Yaskawa INFORM job: DPRINT3D7.JBI

/JOB
//NAME DPRINT3D7
//POS
///NPOS 985,0,0,0,0,0
///TOOL 9
///POSTYPE PULSE
///PULSE
C00000=38331,58153,-103296,76545,-120383,-87250,0
C00001=38829,58071,-103540,76008,-120603,-87388,0
C00002=39135,58069,-103553,75698,-120771,-87432,0
C00003=39547,58102,-103468,75295,-121021,-87464,0
C00004=40049,58223,-103131,74838,-121386,-87436,0
C00005=40275,59096,-100656,75000,-122141,-86754,0
C00006=47985,53725,-116873,64386,-120957,-92528,0
C00007=47675,53509,-117561,64622,-120583,-92677,0
C00008=47512,53337,-118114,64720,-120319,-92811,0
C00009=47414,53155,-118707,64742,-120065,-92966,0
C00010=47387,52969,-119318,64686,-119830,-93137,0
C00011=47431,52787,-119922,64554,-119625,-93316,0
C00012=47549,52614,-120504,64346,-119454,-93499,0
C00013=47574,52593,-120575,64308,-119436,-93523,0
C00014=47628,52527,-120798,64219,-119373,-93594,0
C00015=47840,52374,-121320,63916,-119254,-93772,0
C00016=48067,52268,-121685,63619,-119197,-93907,0
C00017=31263,52363,-120961,59625,-120633,-94164,0
C00018=30956,52566,-120274,60061,-120805,-93930,0
C00019=30684,52688,-119859,60420,-120875,-93775,0
C00020=30370,52784,-119536,60811,-120890,-93639,0
C00021=30027,52848,-119318,61220,-120850,-93528,0
C00022=29664,52879,-119210,61633,-120758,-93444,0
C00023=29293,52875,-119218,62038,-120617,-93392,0
C00024=29245,52869,-119235,62089,-120591,-93390,0
C00025=29099,52864,-119249,62246,-120531,-93372,0
C00026=28731,52813,-119411,62626,-120330,-93365,0
C00027=28447,52743,-119639,62904,-120137,-93388,0
C00028=23605,59262,-99913,71173,-124359,-87087,0
C00029=24011,59446,-99401,70849,-124736,-87010,0
C00030=24270,59629,-98895,70675,-125027,-86912,0
C00031=24478,59852,-98276,70574,-125325,-86774,0
C00032=24629,60106,-97571,70549,-125613,-86602,0
C00033=24674,60248,-97179,70575,-125751,-86501,0
C00034=24716,60482,-96534,70652,-125958,-86328,0
C00035=24702,60771,-95739,70814,-126174,-86103,0
C00036=24621,61063,-94936,71047,-126350,-85865,0
C00037=28498,55123,-112076,85369,-113238,-88875,0
C00038=37681,59282,-100081,77670,-120764,-86229,0
C00039=37996,59009,-100854,77242,-120771,-86495,0
C00040=38275,58852,-101304,76897,-120827,-86663,0
C00041=38591,58743,-101619,76535,-120935,-86797,0
C00042=38928,58687,-101786,76172,-121088,-86891,0
C00043=39106,58685,-101794,75993,-121188,-86918,0
C00044=39389,58708,-101735,75719,-121365,-86940,0
C00045=39717,58789,-101511,75424,-121607,-86921,0
C00046=40017,58920,-101147,75180,-121870,-86858,0
C00047=40209,59050,-100782,75046,-122072,-86781,0
C00048=48256,52888,-119608,63698,-120051,-93341,0
C00049=48323,52793,-119927,63580,-119956,-93441,0
C00050=48337,52781,-119967,63559,-119947,-93454,0
C00051=48383,52725,-120153,63482,-119894,-93514,0
C00052=48503,52640,-120443,63311,-119827,-93613,0
C00053=48657,52567,-120690,63107,-119789,-93704,0
C00054=48843,52511,-120885,62876,-119781,-93786,0
C00055=49053,52474,-121016,62628,-119806,-93852,0
C00056=49530,52439,-121146,62087,-119926,-93955,0
C00057=30578,51713,-123173,60079,-119485,-94678,0
C00058=30592,51957,-122328,60177,-119839,-94445,0
C00059=30557,52051,-122006,60259,-119958,-94350,0
C00060=30547,52064,-121961,60277,-119974,-94336,0
C00061=30518,52123,-121760,60336,-120045,-94277,0
C00062=30431,52212,-121454,60474,-120140,-94179,0
C00063=30313,52291,-121186,60642,-120207,-94088,0
C00064=30163,52358,-120957,60839,-120246,-94002,0
C00065=29988,52410,-120777,61056,-120257,-93927,0
C00066=29796,52445,-120656,61284,-120236,-93866,0
C00067=29593,52462,-120596,61515,-120187,-93820,0
C00068=29386,52460,-120600,61742,-120110,-93791,0
C00069=29358,52457,-120610,61771,-120096,-93790,0
C00070=29234,52452,-120622,61905,-120047,-93776,0
C00071=29027,52424,-120713,62120,-119936,-93772,0
C00072=28832,52377,-120868,62313,-119804,-93789,0
C00073=28655,52311,-121087,62476,-119656,-93826,0
C00074=28506,52230,-121360,62602,-119496,-93883,0
C00075=28262,52031,-122031,62779,-119148,-94040,0
C00076=22525,59894,-98134,72576,-124225,-86409,0
C00077=23013,59805,-98387,72040,-124442,-86560,0
C00078=23209,59804,-98394,71841,-124555,-86594,0
C00079=23405,59836,-98307,71658,-124693,-86602,0
C00080=23465,59857,-98249,71607,-124744,-86596,0
C00081=23613,59925,-98061,71491,-124883,-86567,0
C00082=23766,60034,-97760,71390,-125056,-86508,0
C00083=23890,60167,-97394,71331,-125230,-86427,0
C00084=23981,60318,-96976,71315,-125400,-86325,0
C00085=23998,60372,-96827,71324,-125452,-86286,0
C00086=24026,60515,-96435,71368,-125577,-86181,0
C00087=24020,60684,-95968,71460,-125703,-86049,0
C00088=23975,60851,-95509,71589,-125803,-85913,0
C00089=23899,60999,-95103,71741,-125867,-85785,0
C00090=23790,61133,-94734,71919,-125901,-85664,0
C00091=23657,61244,-94431,72108,-125903,-85556,0
C00092=23222,61486,-93767,72664,-125812,-85295,0
C00093=38158,60313,-97216,77640,-121705,-85464,0
C00094=38179,59892,-98385,77438,-121451,-85805,0
C00095=38226,59733,-98827,77323,-121377,-85939,0
C00096=38312,59585,-99244,77175,-121331,-86071,0
C00097=38351,59542,-99365,77117,-121327,-86112,0
C00098=38467,59441,-99648,76958,-121330,-86209,0
C00099=38632,59347,-99915,76754,-121365,-86309,0
C00100=38817,59282,-100102,76542,-121429,-86388,0
C00101=39014,59248,-100201,76330,-121521,-86444,0
C00102=39081,59248,-100204,76264,-121560,-86455,0
C00103=39251,59262,-100167,76100,-121668,-86468,0
C00104=39442,59310,-100036,75931,-121812,-86457,0
C00105=39615,59387,-99824,75792,-121964,-86420,0
C00106=39764,59489,-99539,75689,-122122,-86359,0
C00107=39882,59612,-99198,75626,-122275,-86278,0
C00108=39967,59750,-98814,75604,-122420,-86180,0
C00109=40106,60176,-97632,75659,-122792,-85861,0
C00110=49445,53618,-117255,62738,-121392,-92853,0
C00111=48956,53536,-117508,63236,-121106,-92850,0
C00112=48781,53486,-117664,63403,-120980,-92868,0
C00113=48758,53476,-117695,63424,-120959,-92873,0
C00114=48651,53442,-117803,63524,-120877,-92888,0
C00115=48502,53371,-118031,63654,-120735,-92930,0
C00116=48381,53287,-118302,63747,-120587,-92989,0
C00117=48292,53192,-118608,63800,-120438,-93063,0
C00118=48241,53092,-118936,63809,-120297,-93148,0
C00119=48228,52989,-119273,63775,-120166,-93242,0
C00120=48242,52939,-119441,63736,-120109,-93291,0
C00121=48106,52817,-119840,63829,-119909,-93386,0
C00122=49490,53423,-117887,62596,-121169,-93036,0
C00123=49557,53418,-117905,62520,-121189,-93050,0
C00124=49691,53409,-117940,62368,-121227,-93081,0
C00125=49826,53399,-117976,62215,-121265,-93111,0
C00126=49900,53394,-117995,62132,-121285,-93127,0
C00127=49913,53392,-117999,62117,-121289,-93130,0
C00128=49925,53391,-118003,62102,-121291,-93133,0
C00129=49938,53390,-118008,62087,-121295,-93137,0
C00130=49951,53389,-118013,62072,-121298,-93140,0
C00131=49964,53388,-118017,62057,-121301,-93143,0
C00132=49977,53386,-118022,62042,-121305,-93146,0
C00133=49990,53385,-118026,62028,-121307,-93150,0
C00134=50003,53384,-118030,62013,-121311,-93153,0
C00135=50016,53382,-118034,61998,-121314,-93156,0
C00136=50030,53381,-118039,61983,-121318,-93159,0
C00137=50043,53380,-118042,61967,-121321,-93162,0
C00138=50056,53379,-118047,61952,-121324,-93165,0
C00139=50068,53378,-118052,61938,-121328,-93169,0
C00140=50080,53376,-118056,61924,-121330,-93172,0
C00141=50093,53375,-118061,61910,-121332,-93175,0
C00142=50105,53374,-118067,61896,-121336,-93178,0
C00143=50111,53373,-118068,61889,-121337,-93179,0
C00144=50120,53368,-118085,61876,-121335,-93186,0
C00145=50164,53345,-118162,61817,-121321,-93213,0
C00146=50208,53322,-118238,61758,-121308,-93241,0
C00147=50243,53302,-118302,61710,-121297,-93265,0
C00148=50270,53287,-118355,61672,-121286,-93283,0
C00149=50290,53273,-118397,61644,-121277,-93298,0
C00150=50310,53260,-118441,61615,-121268,-93313,0
C00151=50331,53247,-118484,61587,-121259,-93328,0
C00152=50351,53234,-118527,61558,-121250,-93343,0
C00153=50371,53221,-118570,61529,-121241,-93358,0
C00154=50385,53212,-118602,61509,-121232,-93369,0
C00155=50399,53202,-118635,61489,-121226,-93380,0
C00156=50413,53192,-118668,61469,-121218,-93391,0
C00157=50425,53182,-118700,61451,-121209,-93402,0
C00158=50438,53173,-118732,61433,-121201,-93413,0
C00159=50450,53163,-118765,61414,-121193,-93424,0
C00160=50463,53153,-118797,61396,-121185,-93435,0
C00161=50475,53143,-118830,61377,-121177,-93446,0
C00162=50488,53134,-118862,61359,-121169,-93457,0
C00163=50499,53125,-118892,61342,-121162,-93466,0
C00164=50509,53116,-118919,61327,-121154,-93475,0
C00165=50519,53108,-118947,61312,-121147,-93484,0
C00166=50526,53101,-118969,61301,-121142,-93491,0
C00167=50535,53094,-118993,61288,-121135,-93500,0
C00168=50543,53086,-119020,61275,-121128,-93508,0
C00169=50552,53078,-119048,61261,-121120,-93518,0
C00170=50546,53069,-119075,61263,-121107,-93524,0
C00171=50540,53060,-119104,61266,-121093,-93531,0
C00172=50534,53051,-119133,61269,-121080,-93538,0
C00173=50527,53042,-119164,61272,-121065,-93546,0
C00174=50520,53033,-119194,61275,-121051,-93553,0
C00175=50513,53023,-119225,61279,-121036,-93560,0
C00176=50506,53014,-119255,61282,-121021,-93568,0
C00177=50499,53005,-119286,61285,-121007,-93575,0
C00178=50492,52996,-119316,61288,-120992,-93583,0
C00179=50485,52986,-119347,61292,-120977,-93590,0
C00180=50478,52977,-119377,61295,-120964,-93598,0
C00181=50470,52968,-119408,61299,-120947,-93605,0
C00182=50461,52958,-119440,61304,-120933,-93613,0
C00183=50453,52948,-119472,61309,-120916,-93620,0
C00184=50444,52938,-119504,61314,-120900,-93628,0
C00185=50432,52927,-119543,61321,-120881,-93636,0
C00186=50421,52915,-119582,61328,-120861,-93646,0
C00187=50409,52903,-119621,61336,-120842,-93655,0
C00188=50397,52891,-119660,61343,-120822,-93664,0
C00189=50385,52879,-119698,61351,-120803,-93673,0
C00190=50373,52867,-119737,61358,-120782,-93682,0
C00191=50359,52855,-119779,61367,-120761,-93692,0
C00192=50344,52841,-119822,61377,-120738,-93701,0
C00193=50326,52826,-119873,61391,-120712,-93713,0
C00194=50303,52808,-119932,61408,-120681,-93726,0
C00195=50280,52790,-119990,61424,-120649,-93739,0
C00196=50258,52773,-120049,61441,-120618,-93752,0
C00197=50231,52753,-120114,61461,-120582,-93766,0
C00198=50191,52726,-120201,61492,-120534,-93784,0
C00199=50166,52711,-120252,61512,-120505,-93795,0
C00200=50160,52710,-120257,61519,-120500,-93795,0
C00201=50148,52707,-120265,61531,-120494,-93796,0
C00202=50136,52704,-120273,61543,-120486,-93797,0
C00203=50124,52702,-120281,61555,-120477,-93797,0
C00204=50112,52699,-120290,61566,-120471,-93798,0
C00205=50100,52697,-120298,61579,-120463,-93798,0
C00206=50089,52694,-120305,61590,-120456,-93799,0
C00207=50079,52692,-120312,61600,-120450,-93799,0
C00208=50068,52690,-120319,61611,-120443,-93800,0
C00209=50057,52688,-120326,61622,-120436,-93800,0
C00210=50045,52686,-120332,61634,-120429,-93800,0
C00211=49900,52663,-120404,61783,-120350,-93799,0
C00212=49755,52641,-120475,61933,-120269,-93798,0
C00213=49610,52619,-120545,62083,-120189,-93797,0
C00214=30191,51747,-123046,60523,-119408,-94589,0
C00215=30111,51679,-123283,60580,-119283,-94644,0
C00216=30030,51611,-123519,60638,-119159,-94700,0
C00217=29986,51574,-123646,60670,-119093,-94730,0
C00218=29979,51568,-123665,60675,-119082,-94734,0
C00219=29971,51563,-123685,60681,-119072,-94738,0
C00220=29964,51558,-123703,60687,-119062,-94742,0
C00221=29957,51552,-123723,60692,-119051,-94747,0
C00222=29949,51547,-123741,60698,-119042,-94751,0
C00223=29942,51541,-123759,60703,-119032,-94756,0
C00224=29935,51536,-123779,60709,-119021,-94760,0
C00225=29927,51530,-123797,60715,-119011,-94765,0
C00226=29920,51525,-123817,60720,-119001,-94769,0
C00227=29913,51519,-123835,60726,-118990,-94773,0
C00228=29905,51514,-123855,60732,-118980,-94777,0
C00229=29898,51509,-123873,60737,-118971,-94781,0
C00230=29891,51504,-123892,60743,-118961,-94785,0
C00231=29884,51499,-123908,60748,-118951,-94789,0
C00232=29877,51494,-123925,60754,-118942,-94793,0
C00233=29869,51489,-123941,60760,-118933,-94797,0
C00234=29866,51487,-123949,60763,-118928,-94799,0
C00235=29852,51484,-123959,60776,-118920,-94800,0
C00236=29791,51472,-124001,60838,-118882,-94803,0
C00237=29730,51460,-124042,60900,-118846,-94807,0
C00238=29679,51450,-124075,60952,-118816,-94809,0
C00239=29638,51443,-124100,60994,-118792,-94811,0
C00240=29605,51438,-124116,61028,-118774,-94811,0
C00241=29572,51433,-124132,61063,-118757,-94812,0
C00242=29539,51429,-124149,61097,-118739,-94812,0
C00243=29506,51424,-124165,61131,-118722,-94812,0
C00244=29473,51419,-124182,61165,-118704,-94813,0
C00245=29449,51416,-124192,61191,-118692,-94812,0
C00246=29424,51413,-124202,61217,-118680,-94812,0
C00247=29400,51410,-124212,61242,-118668,-94812,0
C00248=29376,51407,-124220,61268,-118656,-94810,0
C00249=29352,51405,-124227,61293,-118646,-94810,0
C00250=29328,51403,-124235,61318,-118634,-94809,0
C00251=29305,51400,-124243,61344,-118623,-94808,0
C00252=29281,51398,-124251,61369,-118612,-94807,0
C00253=29257,51396,-124259,61394,-118601,-94806,0
C00254=29235,51394,-124266,61417,-118592,-94805,0
C00255=29215,51392,-124272,61439,-118583,-94804,0
C00256=29195,51390,-124278,61460,-118573,-94803,0
C00257=29179,51389,-124281,61477,-118566,-94802,0
C00258=29161,51388,-124285,61496,-118560,-94801,0
C00259=29142,51387,-124289,61517,-118551,-94799,0
C00260=29122,51385,-124293,61538,-118543,-94798,0
C00261=29101,51393,-124265,61565,-118548,-94787,0
C00262=29086,51399,-124246,61584,-118550,-94780,0
C00263=29071,51404,-124225,61603,-118554,-94772,0
C00264=29055,51410,-124204,61623,-118557,-94764,0
C00265=29040,51416,-124182,61643,-118561,-94756,0
C00266=29025,51422,-124162,61662,-118564,-94748,0
C00267=29009,51428,-124141,61682,-118568,-94740,0
C00268=28994,51434,-124119,61702,-118571,-94732,0
C00269=28979,51440,-124098,61721,-118574,-94724,0
C00270=28963,51446,-124078,61741,-118578,-94716,0
C00271=28948,51451,-124056,61760,-118581,-94708,0
C00272=28932,51458,-124033,61781,-118586,-94699,0
C00273=28917,51465,-124009,61801,-118589,-94690,0
C00274=28901,51472,-123985,61822,-118594,-94682,0
C00275=28884,51479,-123957,61844,-118600,-94671,0
C00276=28865,51488,-123926,61868,-118607,-94660,0
C00277=28846,51497,-123894,61893,-118612,-94648,0
C00278=28828,51506,-123863,61918,-118619,-94637,0
C00279=28809,51515,-123832,61942,-118625,-94626,0
C00280=28791,51524,-123800,61966,-118632,-94614,0
C00281=28772,51532,-123769,61991,-118638,-94603,0
C00282=28752,51543,-123731,62018,-118647,-94590,0
C00283=28732,51554,-123694,62045,-118655,-94577,0
C00284=28706,51569,-123639,62081,-118668,-94557,0
C00285=28680,51584,-123585,62116,-118680,-94538,0
C00286=28654,51600,-123530,62152,-118693,-94520,0
C00287=28628,51615,-123476,62188,-118707,-94500,0
C00288=28597,51635,-123406,62230,-118724,-94476,0
C00289=28555,51667,-123295,62291,-118754,-94440,0
C00290=28555,51673,-123275,62294,-118762,-94433,0
C00291=28554,51679,-123254,62298,-118770,-94427,0
C00292=28554,51685,-123232,62301,-118778,-94422,0
C00293=28553,51691,-123211,62304,-118786,-94415,0
C00294=28553,51697,-123191,62307,-118794,-94409,0
C00295=28553,51703,-123170,62310,-118802,-94404,0
C00296=28552,51708,-123153,62313,-118809,-94398,0
C00297=28552,51713,-123134,62315,-118816,-94393,0
C00298=28552,51718,-123116,62317,-118824,-94388,0
C00299=28553,51724,-123096,62320,-118831,-94383,0
C00300=28559,51761,-122965,62330,-118885,-94346,0
C00301=28570,51831,-122724,62350,-118985,-94278,0
C00302=28581,51902,-122480,62370,-119084,-94211,0
C00303=28587,51937,-122360,62380,-119133,-94177,0
C00304=26988,56207,-108778,66138,-123397,-90126,0
C00305=27559,55476,-110984,65169,-122914,-90833,0
C00306=34385,54484,-114157,79150,-115754,-90039,0
C00307=35133,53863,-116128,78153,-115638,-90720,0
C00308=28153,54774,-113144,64187,-122418,-91528,0
C00309=28772,54099,-115260,63191,-121909,-92212,0
C00310=35909,53269,-118056,77124,-115507,-91394,0
C00311=36715,52701,-119942,76063,-115359,-92059,0
C00312=29489,53589,-116898,62162,-121584,-92777,0
C00313=29679,53591,-116893,61956,-121660,-92805,0
C00314=30389,53528,-117109,61146,-121854,-92975,0
C00315=30449,53516,-117148,61075,-121862,-92995,0
C00316=37553,52159,-121785,74968,-115195,-92717,0
C00317=32557,56236,-108783,60130,-125967,-91111,0
C00318=31344,53310,-117832,59990,-121933,-93322,0
C00319=31411,53289,-117902,59905,-121930,-93352,0
C00320=32489,53643,-116779,58887,-122791,-93223,0
C00321=33235,55545,-110873,59024,-125452,-91789,0
C00322=33580,55212,-111891,58471,-125194,-92120,0
C00323=34127,55436,-111218,57982,-125691,-92047,0
C00324=33632,54047,-115515,57822,-123745,-93081,0
C00325=34746,54472,-114200,56798,-124719,-92936,0
C00326=41514,51531,-124061,70453,-116003,-93828,0
C00327=42611,51965,-122576,69442,-116893,-93495,0
C00328=35832,54919,-112836,55815,-125714,-92788,0
C00329=45678,52142,-122048,66179,-118202,-93704,0
C00330=45685,52643,-120356,66395,-118810,-93209,0
C00331=45693,53257,-118329,66662,-119525,-92621,0
C00332=45700,53794,-116593,66900,-120126,-92121,0
C00333=44762,54321,-114897,68151,-120297,-91501,0
C00334=44638,51679,-123626,67113,-117264,-94046,0
C00335=43562,51238,-125158,68100,-116350,-94385,0
C00336=43855,54873,-113154,69373,-120456,-90871,0
C00337=42976,55449,-111365,70566,-120600,-90230,0
C00338=42574,51681,-123560,69364,-116551,-93790,0
C00339=41623,52167,-121858,70596,-116757,-93166,0
C00340=42126,56052,-109528,71730,-120734,-89579,0
C00341=41304,56680,-107641,72868,-120856,-88917,0
C00342=40707,52678,-120113,71792,-116945,-92533,0
C00343=39824,53213,-118325,72955,-117117,-91892,0
C00344=40507,57334,-105705,73979,-120965,-88245,0
C00345=39896,57870,-104139,74839,-121043,-87706,0
C00346=39759,57838,-104230,74965,-120944,-87714,0
C00347=39709,57834,-104241,75013,-120914,-87710,0
C00348=38973,53774,-116493,74084,-117275,-91241,0
C00349=38152,54361,-114618,75181,-117415,-90581,0
C00350=38839,57797,-104329,75882,-120413,-87619,0
C00351=38784,57798,-104326,75937,-120383,-87610,0
C00352=38125,57905,-104004,76648,-120097,-87430,0
C00353=38000,57947,-103882,76792,-120057,-87378,0
C00354=37361,54974,-112698,76248,-117543,-89913,0
C00355=36597,55613,-110732,77286,-117655,-89235,0
C00356=37083,57698,-104582,77613,-119379,-87467,0
C00357=36088,57176,-106077,78410,-118484,-87789,0
C00358=35597,55333,-111561,78209,-116954,-89374,0
C00359=35382,55525,-110973,78501,-116984,-89174,0
C00360=34626,55201,-111945,79159,-116380,-89388,0
C00361=35067,56678,-107520,79250,-117606,-88101,0
C00362=34023,56202,-108911,80133,-116743,-88407,0
C00363=26988,56207,-108778,66138,-123397,-90126,0
C00364=26438,56968,-106524,67097,-123870,-89408,0
C00365=32953,55749,-110251,81058,-115896,-88704,0
C00366=31858,55317,-111539,82026,-115065,-88994,0
C00367=25909,57758,-104221,68046,-124333,-88678,0
C00368=25407,58565,-101904,68972,-124779,-87946,0
C00369=25677,58848,-101106,68834,-125167,-87771,0
C00370=25959,59324,-99770,68784,-125726,-87448,0
C00371=26059,59657,-98840,68852,-126061,-87208,0
C00372=30505,54262,-114777,83075,-113747,-89879,0
C00373=30483,54351,-114498,83125,-113791,-89790,0
C00374=30737,54907,-112777,83035,-114252,-89276,0
C00375=36475,52909,-119246,76394,-115443,-91819,0
C00376=39287,53519,-117321,73649,-117178,-91527,0
C00377=37677,52791,-119666,75075,-115836,-92070,0
C00378=33817,55911,-109778,58572,-126132,-91613,0
C00379=41548,52077,-122164,70640,-116630,-93251,0
C00380=38066,54265,-114919,75233,-117295,-90662,0
C00381=37534,52314,-121259,75046,-115335,-92550,0
C00382=37535,52252,-121281,75054,-115355,-92528,0
C00383=23394,59896,-98012,71737,-124791,-86493,0
C00384=23307,59866,-98096,71810,-124718,-86502,0
C00385=23275,59856,-98122,71837,-124691,-86504,0
C00386=23229,59845,-98154,71878,-124656,-86506,0
C00387=23180,59837,-98176,71923,-124621,-86504,0
C00388=23118,59828,-98200,71981,-124579,-86500,0
C00389=23054,59822,-98215,72044,-124537,-86494,0
C00390=22961,59823,-98212,72138,-124483,-86478,0
C00391=22921,59825,-98206,72180,-124462,-86470,0
C00392=22873,59829,-98192,72231,-124436,-86458,0
C00393=22786,59845,-98148,72326,-124398,-86431,0
C00394=22744,59854,-98121,72373,-124381,-86417,0
C00395=22700,59867,-98087,72423,-124364,-86401,0
C00396=22631,59892,-98014,72505,-124343,-86369,0
C00397=22541,59936,-97893,72617,-124323,-86320,0
C00398=22471,59982,-97763,72710,-124316,-86272,0
C00399=22404,60033,-97623,72802,-124313,-86221,0
C00400=22346,60090,-97463,72888,-124321,-86167,0
C00401=22292,60151,-97293,72971,-124335,-86110,0
C00402=22281,60166,-97251,72989,-124340,-86096,0
C00403=22248,60218,-97109,73047,-124357,-86051,0
C00404=22210,60287,-96917,73119,-124385,-85991,0
C00405=22180,60370,-96689,73188,-124427,-85921,0
C00406=22165,60435,-96507,73236,-124466,-85868,0
C00407=22160,60475,-96397,73260,-124491,-85836,0
C00408=22158,60512,-96296,73280,-124517,-85807,0
C00409=22158,60589,-96084,73317,-124572,-85747,0
C00410=22162,60631,-95969,73333,-124605,-85715,0
C00411=22168,60666,-95875,73344,-124633,-85689,0
C00412=22186,60745,-95657,73365,-124701,-85631,0
C00413=22205,60799,-95509,73372,-124751,-85592,0
C00414=22228,60849,-95372,73374,-124801,-85557,0
C00415=22247,60890,-95261,73375,-124841,-85529,0
C00416=22269,60927,-95159,73371,-124881,-85504,0
C00417=22309,60984,-95005,73359,-124945,-85467,0
C00418=22337,61021,-94903,73350,-124989,-85443,0
C00419=22368,61055,-94812,73336,-125033,-85422,0
C00420=22417,61101,-94686,73310,-125095,-85395,0
C00421=22453,61133,-94599,73290,-125140,-85376,0
C00422=22491,61162,-94520,73266,-125184,-85360,0
C00423=22546,61197,-94426,73229,-125243,-85343,0
C00424=22589,61223,-94356,73199,-125287,-85330,0
C00425=22634,61245,-94296,73165,-125332,-85321,0
C00426=22654,61253,-94273,73150,-125349,-85318,0
C00427=22740,61286,-94185,73081,-125426,-85307,0
C00428=22808,61305,-94135,73022,-125481,-85304,0
C00429=22900,61322,-94090,72940,-125549,-85307,0
C00430=22969,61328,-94075,72874,-125596,-85315,0
C00431=23064,61328,-94075,72780,-125654,-85331,0
C00432=23119,61323,-94088,72723,-125685,-85344,0
C00433=23209,61312,-94120,72628,-125733,-85368,0
C00434=23286,61294,-94170,72541,-125767,-85396,0
C00435=23362,61271,-94234,72454,-125797,-85426,0
C00436=23434,61239,-94320,72366,-125819,-85463,0
C00437=23504,61204,-94418,72278,-125835,-85502,0
C00438=23568,61160,-94538,72192,-125842,-85547,0
C00439=23629,61113,-94667,72107,-125844,-85593,0
C00440=23683,61059,-94815,72027,-125837,-85644,0
C00441=23733,61002,-94971,71948,-125826,-85696,0
C00442=23774,60940,-95141,71875,-125805,-85751,0
C00443=23810,60876,-95317,71806,-125779,-85807,0
C00444=23835,60815,-95486,71750,-125747,-85859,0
C00445=23860,60739,-95694,71687,-125705,-85921,0
C00446=23871,60669,-95887,71640,-125659,-85977,0
C00447=23876,60622,-96015,71612,-125627,-86014,0
C00448=23878,60597,-96082,71597,-125610,-86033,0
C00449=23876,60526,-96278,71563,-125554,-86087,0
C00450=23870,60468,-96439,71539,-125507,-86131,0
C00451=23853,60385,-96668,71515,-125434,-86193,0
C00452=23834,60325,-96830,71505,-125377,-86235,0
C00453=23799,60249,-97041,71502,-125298,-86288,0
C00454=23766,60193,-97195,71507,-125236,-86326,0
C00455=23714,60125,-97384,71526,-125153,-86370,0
C00456=23667,60074,-97523,71548,-125087,-86401,0
C00457=23601,60017,-97682,71587,-125004,-86435,0
C00458=23541,59974,-97800,71625,-124937,-86458,0
C00459=23468,59932,-97916,71679,-124861,-86478,0
C00460=23393,59890,-98030,71734,-124787,-86498,0
C00461=35331,54513,-113922,78210,-116284,-90036,0
C00462=36294,54920,-112685,77364,-117050,-89763,0
C00463=40946,51800,-122908,71212,-116196,-93384,0
C00464=33828,55886,-109704,58589,-126201,-91572,0
C00465=35386,54467,-114067,78137,-116276,-90086,0
C00466=35602,55200,-111812,78184,-116919,-89424,0
C00467=36475,55591,-110642,77434,-117637,-89168,0
C00468=42173,51768,-123052,69869,-116605,-93562,0
C00469=33599,55210,-111743,58490,-125297,-92062,0
C00470=34231,54631,-113535,79390,-115843,-89806,0
C00471=35132,54999,-112418,78593,-116543,-89557,0
C00472=34897,55209,-111772,78911,-116575,-89336,0
C00473=35366,55411,-111167,78505,-116951,-89203,0
C00474=35548,55248,-111666,78257,-116925,-89373,0
C00475=36108,54971,-112524,77576,-116998,-89694,0
C00476=34832,55467,-110986,57257,-126113,-92098,0
C00477=36977,53692,-116543,53945,-124582,-93918,0
C00478=39300,53750,-116408,73761,-117469,-91225,0
C00479=44308,56417,-108340,69642,-122190,-89529,0
C00480=34851,55449,-111041,79046,-116720,-89110,0
C00481=32913,57439,-105115,81710,-116938,-87125,0
C00482=36071,54502,-113971,77439,-116627,-90128,0
C00483=40136,51777,-122967,72078,-115873,-93316,0
C00484=48422,53258,-118219,63727,-120668,-92946,0
C00485=48439,53269,-118186,63714,-120687,-92938,0
C00486=48516,53313,-118044,63650,-120769,-92909,0
C00487=48581,53344,-117946,63594,-120831,-92892,0
C00488=48673,53380,-117832,63510,-120910,-92873,0
C00489=48745,53403,-117759,63442,-120965,-92863,0
C00490=48847,53429,-117677,63342,-121035,-92855,0
C00491=48909,53441,-117639,63281,-121073,-92854,0
C00492=49019,53461,-117580,63169,-121138,-92854,0
C00493=49115,53471,-117549,63069,-121186,-92859,0
C00494=49212,53478,-117530,62966,-121232,-92869,0
C00495=49309,53478,-117531,62859,-121269,-92883,0
C00496=49406,53475,-117544,62752,-121303,-92901,0
C00497=49502,53466,-117577,62642,-121327,-92925,0
C00498=49596,53453,-117621,62533,-121346,-92952,0
C00499=49685,53434,-117685,62425,-121357,-92983,0
C00500=49773,53412,-117759,62319,-121362,-93017,0
C00501=49854,53384,-117850,62216,-121359,-93054,0
C00502=49931,53354,-117952,62117,-121350,-93095,0
C00503=49995,53321,-118057,62032,-121332,-93133,0
C00504=50066,53280,-118194,61933,-121307,-93182,0
C00505=50120,53239,-118330,61854,-121275,-93228,0
C00506=50153,53211,-118423,61804,-121252,-93259,0
C00507=50170,53196,-118472,61779,-121238,-93275,0
C00508=50210,53150,-118623,61712,-121196,-93323,0
C00509=50239,53111,-118749,61661,-121157,-93363,0
C00510=50271,53054,-118939,61599,-121095,-93419,0
C00511=50286,53011,-119079,61562,-121046,-93461,0
C00512=50294,52953,-119271,61525,-120974,-93515,0
C00513=50293,52909,-119417,61506,-120915,-93555,0
C00514=50278,52851,-119606,61495,-120836,-93606,0
C00515=50259,52807,-119752,61495,-120772,-93643,0
C00516=50222,52753,-119932,61510,-120688,-93688,0
C00517=50184,52710,-120073,61532,-120618,-93722,0
C00518=50126,52661,-120235,61572,-120534,-93759,0
C00519=50071,52622,-120364,61615,-120463,-93787,0
C00520=49995,52579,-120504,61679,-120381,-93815,0
C00521=49966,52565,-120551,61703,-120352,-93824,0
C00522=49923,52545,-120615,61742,-120311,-93836,0
C00523=49874,52527,-120674,61787,-120271,-93845,0
C00524=49812,52505,-120746,61845,-120220,-93856,0
C00525=49745,52484,-120814,61909,-120169,-93866,0
C00526=49642,52460,-120892,62011,-120102,-93873,0
C00527=49597,52451,-120923,62057,-120073,-93876,0
C00528=49541,52441,-120954,62115,-120041,-93876,0
C00529=49435,52428,-120996,62225,-119987,-93873,0
C00530=49382,52422,-121012,62280,-119961,-93870,0
C00531=49326,52418,-121024,62340,-119937,-93866,0
C00532=49233,52416,-121029,62441,-119902,-93854,0
C00533=49107,52419,-121015,62582,-119862,-93833,0
C00534=48999,52429,-120979,62706,-119837,-93807,0
C00535=48893,52443,-120930,62828,-119818,-93779,0
C00536=48793,52463,-120859,62948,-119809,-93744,0
C00537=48695,52486,-120779,63067,-119805,-93708,0
C00538=48674,52493,-120756,63093,-119806,-93699,0
C00539=48605,52516,-120676,63179,-119811,-93667,0
C00540=48520,52548,-120566,63288,-119822,-93623,0
C00541=48436,52591,-120419,63400,-119848,-93570,0
C00542=48379,52628,-120295,63480,-119873,-93527,0
C00543=48349,52651,-120217,63523,-119893,-93501,0
C00544=48325,52674,-120142,63561,-119911,-93476,0
C00545=48278,52721,-119982,63634,-119953,-93424,0
C00546=48257,52748,-119891,63669,-119980,-93396,0
C00547=48243,52771,-119816,63695,-120004,-93372,0
C00548=48216,52825,-119636,63750,-120060,-93317,0
C00549=48205,52863,-119509,63780,-120104,-93279,0
C00550=48200,52901,-119386,63802,-120149,-93244,0
C00551=48198,52931,-119286,63819,-120184,-93215,0
C00552=48201,52960,-119189,63830,-120222,-93188,0
C00553=48212,53006,-119039,63839,-120282,-93147,0
C00554=48222,53037,-118938,63843,-120323,-93119,0
C00555=48236,53066,-118842,63841,-120365,-93095,0
C00556=48264,53108,-118704,63830,-120427,-93060,0
C00557=48285,53138,-118608,63821,-120471,-93035,0
C00558=48311,53167,-118515,63806,-120515,-93013,0
C00559=48352,53204,-118395,63778,-120575,-92985,0
C00560=48365,53215,-118360,63770,-120594,-92977,0
C00561=48397,53262,-118207,63756,-120662,-92938,0
C00562=30428,52147,-121485,60486,-120164,-94162,0
C00563=30434,52142,-121505,60477,-120158,-94167,0
C00564=30467,52107,-121623,60424,-120122,-94205,0
C00565=30508,52051,-121815,60353,-120058,-94264,0
C00566=30527,52011,-121952,60313,-120009,-94305,0
C00567=30542,51955,-122141,60270,-119936,-94359,0
C00568=30545,51923,-122253,60253,-119891,-94391,0
C00569=30543,51869,-122436,60229,-119816,-94442,0
C00570=30529,51823,-122595,60223,-119745,-94484,0
C00571=30509,51777,-122753,60224,-119674,-94525,0
C00572=30475,51733,-122906,60241,-119600,-94563,0
C00573=30436,51690,-123054,60265,-119526,-94599,0
C00574=30384,51649,-123192,60304,-119451,-94630,0
C00575=30326,51611,-123325,60350,-119377,-94659,0
C00576=30257,51576,-123445,60410,-119304,-94683,0
C00577=30183,51543,-123557,60477,-119233,-94705,0
C00578=30100,51515,-123654,60555,-119166,-94720,0
C00579=30013,51490,-123741,60640,-119102,-94733,0
C00580=29919,51470,-123810,60734,-119042,-94740,0
C00581=29823,51452,-123870,60833,-118986,-94744,0
C00582=29722,51441,-123909,60939,-118936,-94741,0
C00583=29654,51435,-123928,61011,-118907,-94738,0
C00584=29619,51432,-123938,61049,-118890,-94735,0
C00585=29515,51428,-123949,61162,-118851,-94725,0
C00586=29430,51427,-123951,61256,-118822,-94715,0
C00587=29306,51431,-123935,61394,-118787,-94694,0
C00588=29217,51437,-123911,61495,-118768,-94675,0
C00589=29101,51451,-123858,61630,-118750,-94645,0
C00590=29015,51466,-123805,61731,-118742,-94618,0
C00591=28909,51490,-123718,61860,-118742,-94579,0
C00592=28829,51513,-123638,61957,-118747,-94546,0
C00593=28737,51546,-123520,62074,-118763,-94501,0
C00594=28668,51576,-123415,62164,-118781,-94462,0
C00595=28594,51617,-123271,62264,-118813,-94411,0
C00596=28538,51653,-123144,62341,-118845,-94367,0
C00597=28484,51700,-122980,62422,-118890,-94314,0
C00598=28467,51717,-122922,62449,-118908,-94294,0
C00599=28445,51742,-122834,62485,-118934,-94267,0
C00600=28428,51769,-122741,62516,-118965,-94238,0
C00601=28408,51803,-122623,62553,-119004,-94202,0
C00602=28393,51839,-122499,62586,-119048,-94165,0
C00603=28384,51892,-122317,62620,-119116,-94112,0
C00604=28383,51915,-122239,62632,-119146,-94089,0
C00605=28385,51943,-122144,62643,-119184,-94062,0
C00606=28398,51994,-121970,62651,-119256,-94015,0
C00607=28407,52018,-121886,62652,-119292,-93992,0
C00608=28420,52044,-121798,62650,-119331,-93969,0
C00609=28440,52073,-121701,62641,-119375,-93944,0
C00610=28456,52094,-121631,62633,-119409,-93927,0
C00611=28502,52141,-121470,62604,-119487,-93887,0
C00612=28561,52186,-121321,62560,-119567,-93853,0
C00613=28626,52229,-121177,62509,-119645,-93821,0
C00614=28701,52267,-121049,62444,-119724,-93795,0
C00615=28781,52304,-120927,62373,-119799,-93772,0
C00616=28871,52335,-120823,62289,-119872,-93755,0
C00617=28964,52364,-120729,62200,-119943,-93742,0
C00618=28987,52369,-120711,62177,-119959,-93740,0
C00619=29076,52388,-120648,62088,-120016,-93735,0
C00620=29167,52403,-120599,61995,-120067,-93735,0
C00621=29223,52410,-120579,61937,-120096,-93736,0
C00622=29274,52415,-120564,61883,-120120,-93740,0
C00623=29386,52422,-120542,61763,-120169,-93749,0
C00624=29465,52423,-120540,61676,-120199,-93760,0
C00625=29543,52421,-120546,61590,-120225,-93773,0
C00626=29603,52419,-120553,61524,-120244,-93784,0
C00627=29659,52415,-120568,61460,-120258,-93796,0
C00628=29702,52411,-120584,61410,-120267,-93806,0
C00629=29812,52397,-120633,61283,-120288,-93836,0
C00630=29904,52380,-120692,61174,-120297,-93866,0
C00631=30007,52355,-120775,61049,-120300,-93903,0
C00632=30087,52331,-120860,60948,-120296,-93939,0
C00633=30179,52297,-120974,60832,-120283,-93983,0
C00634=30247,52267,-121080,60742,-120265,-94022,0
C00635=30322,52226,-121218,60641,-120235,-94072,0
C00636=30376,52190,-121342,60564,-120204,-94114,0
C00637=30442,52147,-121485,60471,-120168,-94163,0
C00638=25183,55522,-110657,67769,-121953,-90344,0
C00639=36362,52582,-120147,76424,-115182,-92059,0
C00640=39661,59488,-99412,75825,-122113,-86283,0
C00641=39593,59449,-99522,75876,-122046,-86305,0
C00642=39522,59413,-99620,75931,-121981,-86323,0
C00643=39445,59385,-99696,75995,-121916,-86334,0
C00644=39394,59369,-99740,76039,-121876,-86340,0
C00645=39366,59362,-99761,76062,-121855,-86342,0
C00646=39285,59345,-99806,76136,-121796,-86344,0
C00647=39218,59334,-99835,76199,-121750,-86343,0
C00648=39119,59326,-99854,76294,-121686,-86334,0
C00649=39046,59327,-99852,76366,-121644,-86323,0
C00650=38950,59335,-99826,76466,-121593,-86302,0
C00651=38877,59348,-99790,76544,-121559,-86282,0
C00652=38785,59372,-99721,76646,-121521,-86249,0
C00653=38715,59396,-99651,76726,-121497,-86220,0
C00654=38632,59435,-99542,76825,-121473,-86176,0
C00655=38568,59471,-99438,76905,-121459,-86138,0
C00656=38496,59522,-99294,76997,-121451,-86086,0
C00657=38441,59569,-99162,77072,-121449,-86040,0
C00658=38384,59631,-98987,77156,-121454,-85982,0
C00659=38365,59654,-98923,77184,-121459,-85961,0
C00660=38340,59689,-98827,77224,-121466,-85930,0
C00661=38319,59726,-98724,77261,-121476,-85897,0
C00662=38293,59773,-98591,77307,-121491,-85855,0
C00663=38270,59824,-98450,77351,-121511,-85811,0
C00664=38248,59899,-98240,77406,-121545,-85747,0
C00665=38240,59932,-98147,77428,-121561,-85719,0
C00666=38233,59973,-98035,77452,-121583,-85686,0
C00667=38229,60048,-97827,77488,-121628,-85626,0
C00668=38229,60084,-97725,77504,-121652,-85596,0
C00669=38232,60123,-97617,77518,-121678,-85566,0
C00670=38240,60167,-97496,77530,-121711,-85532,0
C00671=38247,60199,-97409,77537,-121735,-85508,0
C00672=38270,60273,-97205,77546,-121794,-85452,0
C00673=38304,60344,-97009,77543,-121861,-85400,0
C00674=38344,60413,-96818,77535,-121929,-85351,0
C00675=38393,60477,-96642,77514,-121999,-85307,0
C00676=38447,60539,-96472,77489,-122071,-85266,0
C00677=38510,60594,-96322,77451,-122145,-85231,0
C00678=38577,60647,-96180,77409,-122218,-85200,0
C00679=38594,60657,-96151,77397,-122236,-85194,0
C00680=38660,60695,-96048,77349,-122300,-85174,0
C00681=38728,60727,-95962,77296,-122362,-85159,0
C00682=38771,60743,-95919,77262,-122399,-85152,0
C00683=38811,60755,-95886,77229,-122431,-85148,0
C00684=38899,60778,-95823,77153,-122500,-85143,0
C00685=38961,60789,-95796,77097,-122545,-85144,0
C00686=39024,60795,-95780,77038,-122588,-85148,0
C00687=39072,60799,-95769,76993,-122621,-85152,0
C00688=39118,60799,-95770,76948,-122648,-85159,0
C00689=39154,60798,-95775,76913,-122670,-85166,0
C00690=39245,60790,-95798,76819,-122722,-85185,0
C00691=39323,60775,-95840,76736,-122760,-85209,0
C00692=39412,60752,-95907,76639,-122800,-85241,0
C00693=39483,60725,-95982,76557,-122825,-85273,0
C00694=39565,60686,-96090,76459,-122852,-85315,0
C00695=39627,60649,-96194,76381,-122865,-85355,0
C00696=39698,60598,-96335,76288,-122876,-85405,0
C00697=39751,60551,-96466,76215,-122877,-85451,0
C00698=39810,60487,-96642,76127,-122871,-85510,0
C00699=39846,60440,-96772,76071,-122862,-85552,0
C00700=39894,60362,-96988,75988,-122839,-85621,0
C00701=39920,60306,-97144,75937,-122818,-85669,0
C00702=39947,60227,-97364,75873,-122782,-85737,0
C00703=39958,60179,-97496,75841,-122756,-85776,0
C00704=39972,60101,-97713,75792,-122711,-85841,0
C00705=39974,60031,-97906,75758,-122667,-85896,0
C00706=39971,59962,-98099,75730,-122617,-85951,0
C00707=39957,59893,-98289,75713,-122563,-86003,0
C00708=39938,59826,-98475,75701,-122506,-86054,0
C00709=39908,59761,-98655,75702,-122445,-86101,0
C00710=39873,59699,-98829,75708,-122382,-86146,0
C00711=39858,59679,-98885,75714,-122359,-86160,0
C00712=39829,59640,-98990,75726,-122315,-86186,0
C00713=39780,59585,-99145,75750,-122248,-86224,0
C00714=39724,59536,-99280,75784,-122183,-86254,0
C00715=39665,59469,-99466,75813,-122102,-86299,0
C00716=39665,59415,-99488,75823,-122118,-86281,0
C00717=23831,60832,-95318,71801,-125814,-85787,0
C00718=23834,60823,-95341,71793,-125810,-85794,0
C00719=23856,60761,-95510,71740,-125776,-85845,0
C00720=23876,60680,-95734,71679,-125727,-85911,0
C00721=23883,60617,-95906,71640,-125684,-85960,0
C00722=23885,60533,-96137,71596,-125622,-86025,0
C00723=23878,60473,-96301,71572,-125573,-86070,0
C00724=23858,60379,-96560,71546,-125489,-86139,0
C00725=23844,60334,-96683,71537,-125448,-86172,0
C00726=23819,60267,-96869,71528,-125381,-86220,0
C00727=23784,60203,-97045,71532,-125312,-86263,0
C00728=23744,60141,-97214,71541,-125242,-86304,0
C00729=23695,60085,-97369,71563,-125169,-86339,0
C00730=23641,60031,-97517,71591,-125097,-86371,0
C00731=23580,59984,-97646,71629,-125026,-86397,0
C00732=23515,59941,-97765,71673,-124955,-86420,0
C00733=23444,59905,-97863,71727,-124886,-86435,0
C00734=23371,59874,-97950,71786,-124819,-86448,0
C00735=23293,59850,-98013,71853,-124756,-86453,0
C00736=23214,59832,-98064,71925,-124695,-86454,0
C00737=23132,59822,-98089,72003,-124641,-86448,0
C00738=23050,59817,-98102,72083,-124588,-86438,0
C00739=22967,59821,-98090,72168,-124543,-86421,0
C00740=22886,59830,-98066,72255,-124502,-86401,0
C00741=22845,59836,-98046,72299,-124483,-86388,0
C00742=22792,59846,-98020,72357,-124459,-86372,0
C00743=22738,59860,-97979,72419,-124439,-86352,0
C00744=22687,59877,-97931,72479,-124421,-86330,0
C00745=22633,59898,-97874,72543,-124405,-86305,0
C00746=22586,59919,-97813,72601,-124394,-86280,0
C00747=22541,59945,-97742,72658,-124386,-86253,0
C00748=22490,59976,-97657,72724,-124379,-86221,0
C00749=22449,60005,-97574,72780,-124375,-86191,0
C00750=22412,60037,-97486,72832,-124378,-86160,0
C00751=22366,60079,-97370,72898,-124381,-86120,0
C00752=22335,60113,-97275,72946,-124388,-86088,0
C00753=22307,60150,-97172,72992,-124398,-86055,0
C00754=22270,60202,-97029,73054,-124414,-86008,0
C00755=22248,60240,-96923,73095,-124428,-85975,0
C00756=22229,60281,-96811,73133,-124447,-85940,0
C00757=22204,60341,-96644,73188,-124475,-85889,0
C00758=22191,60381,-96533,73220,-124497,-85855,0
C00759=22183,60424,-96416,73249,-124522,-85821,0
C00760=22173,60476,-96272,73283,-124555,-85779,0
C00761=22168,60532,-96119,73316,-124591,-85734,0
C00762=22171,60613,-95897,73352,-124651,-85672,0
C00763=22174,60647,-95805,73366,-124676,-85647,0
C00764=22180,60686,-95698,73379,-124709,-85618,0
C00765=22190,60727,-95584,73389,-124744,-85587,0
C00766=22206,60782,-95433,73401,-124793,-85547,0
C00767=22225,60837,-95282,73408,-124844,-85508,0
C00768=22273,60929,-95033,73405,-124938,-85445,0
C00769=22305,60980,-94893,73399,-124994,-85411,0
C00770=22317,60995,-94854,73394,-125012,-85402,0
C00771=22359,61043,-94723,73376,-125072,-85372,0
C00772=22418,61102,-94561,73347,-125150,-85336,0
C00773=22433,61115,-94528,73338,-125168,-85329,0
C00774=22484,61155,-94420,73307,-125228,-85307,0
C00775=22554,61203,-94289,73261,-125305,-85282,0
C00776=22630,61243,-94182,73206,-125380,-85264,0
C00777=22709,61278,-94087,73145,-125453,-85250,0
C00778=22729,61285,-94068,73128,-125472,-85249,0
C00779=22791,61304,-94019,73076,-125523,-85245,0
C00780=22858,61320,-93974,73018,-125576,-85244,0
C00781=22876,61324,-93963,73002,-125590,-85244,0
C00782=22920,61329,-93950,72961,-125620,-85248,0
C00783=22963,61332,-93942,72920,-125649,-85253,0
C00784=23049,61334,-93939,72835,-125704,-85266,0
C00785=23096,61331,-93947,72788,-125730,-85277,0
C00786=23136,61326,-93960,72745,-125752,-85287,0
C00787=23224,61312,-94000,72650,-125796,-85314,0
C00788=23285,61296,-94045,72582,-125821,-85336,0
C00789=23342,61276,-94098,72515,-125843,-85361,0
C00790=23387,61260,-94143,72462,-125859,-85381,0
C00791=23428,61241,-94195,72412,-125870,-85402,0
C00792=23457,61226,-94236,72375,-125877,-85419,0
C00793=23534,61181,-94359,72275,-125891,-85467,0
C00794=23594,61137,-94481,72193,-125896,-85512,0
C00795=23660,61079,-94639,72097,-125893,-85567,0
C00796=23709,61027,-94783,72022,-125884,-85616,0
C00797=23761,60960,-94967,71936,-125867,-85676,0
C00798=23797,60900,-95132,71869,-125844,-85729,0
C00799=23838,60825,-95335,71791,-125813,-85793,0
C00800=35332,54454,-113945,78218,-116301,-90015,0
C00801=36294,54861,-112707,77372,-117067,-89742,0
C00802=40946,51737,-122931,71220,-116218,-93362,0
C00803=33828,55829,-109726,58601,-126228,-91554,0
C00804=35386,54408,-114089,78145,-116292,-90065,0
C00805=35602,55142,-111834,78192,-116935,-89403,0
C00806=36475,55534,-110664,77442,-117653,-89148,0
C00807=42174,51704,-123075,69877,-116629,-93541,0
C00808=33600,55152,-111765,58501,-125325,-92044,0
C00809=34231,54572,-113557,79398,-115858,-89785,0
C00810=35133,54941,-112440,78601,-116559,-89536,0
C00811=34898,55151,-111794,78919,-116591,-89316,0
C00812=35366,55353,-111189,78513,-116967,-89183,0
C00813=35548,55190,-111688,78265,-116942,-89353,0
C00814=36108,54913,-112546,77584,-117015,-89673,0
C00815=34832,55409,-111009,57268,-126141,-92080,0
C00816=36963,53643,-116530,53978,-124624,-93889,0
C00817=39300,53691,-116430,73769,-117489,-91204,0
C00818=44279,56342,-108418,69675,-122178,-89522,0
C00819=34851,55391,-111063,79054,-116735,-89090,0
C00820=32925,57370,-105176,81701,-116951,-87118,0
C00821=36071,54444,-113993,77447,-116644,-90107,0
C00822=40136,51714,-122990,72085,-115895,-93295,0
C00823=48476,53281,-117971,63718,-120815,-92857,0
C00824=48534,53311,-117879,63668,-120872,-92840,0
C00825=48598,53340,-117786,63612,-120931,-92824,0
C00826=48615,53347,-117762,63596,-120946,-92819,0
C00827=48661,53363,-117714,63553,-120983,-92812,0
C00828=48707,53377,-117670,63510,-121018,-92807,0
C00829=48802,53402,-117591,63418,-121084,-92799,0
C00830=48855,53413,-117556,63366,-121118,-92797,0
C00831=48901,53421,-117531,63318,-121145,-92797,0
C00832=49007,53437,-117483,63210,-121205,-92799,0
C00833=49083,53444,-117462,63130,-121242,-92804,0
C00834=49157,53448,-117452,63051,-121275,-92813,0
C00835=49216,53451,-117445,62988,-121300,-92820,0
C00836=49272,53450,-117448,62927,-121321,-92829,0
C00837=49312,53449,-117453,62881,-121335,-92837,0
C00838=49422,53442,-117478,62757,-121368,-92860,0
C00839=49514,53431,-117516,62652,-121389,-92884,0
C00840=49619,53413,-117577,62527,-121407,-92918,0
C00841=49703,53393,-117644,62426,-121414,-92949,0
C00842=49798,53365,-117736,62308,-121416,-92989,0
C00843=49873,53337,-117829,62212,-121409,-93026,0
C00844=49958,53299,-117954,62100,-121393,-93074,0
C00845=50018,53266,-118063,62019,-121375,-93113,0
C00846=50088,53220,-118216,61920,-121343,-93166,0
C00847=50133,53182,-118339,61852,-121312,-93207,0
C00848=50184,53129,-118514,61770,-121263,-93263,0
C00849=50213,53089,-118643,61719,-121224,-93303,0
C00850=50248,53024,-118859,61650,-121153,-93368,0
C00851=50260,52992,-118964,61621,-121118,-93399,0
C00852=50273,52942,-119128,61583,-121058,-93447,0
C00853=50274,52892,-119293,61558,-120995,-93493,0
C00854=50268,52842,-119457,61540,-120928,-93537,0
C00855=50249,52793,-119618,61538,-120858,-93579,0
C00856=50224,52745,-119776,61543,-120787,-93620,0
C00857=50186,52699,-119928,61563,-120713,-93656,0
C00858=50143,52654,-120076,61590,-120638,-93691,0
C00859=50088,52612,-120212,61631,-120565,-93721,0
C00860=50027,52573,-120343,61679,-120492,-93748,0
C00861=49956,52537,-120458,61741,-120421,-93771,0
C00862=49880,52504,-120566,61808,-120351,-93790,0
C00863=49797,52476,-120657,61888,-120286,-93803,0
C00864=49709,52451,-120738,61972,-120222,-93813,0
C00865=49616,52432,-120800,62066,-120165,-93818,0
C00866=49521,52415,-120853,62163,-120110,-93819,0
C00867=49472,52409,-120874,62214,-120084,-93818,0
C00868=49408,52401,-120899,62281,-120051,-93816,0
C00869=49338,52395,-120916,62355,-120020,-93811,0
C00870=49271,52392,-120923,62427,-119993,-93804,0
C00871=49199,52391,-120928,62506,-119965,-93794,0
C00872=49133,52392,-120922,62580,-119943,-93784,0
C00873=49067,52395,-120907,62654,-119926,-93770,0
C00874=48991,52401,-120888,62740,-119906,-93754,0
C00875=48927,52408,-120861,62814,-119894,-93737,0
C00876=48867,52418,-120826,62885,-119885,-93719,0
C00877=48790,52432,-120777,62976,-119875,-93694,0
C00878=48734,52445,-120733,63043,-119872,-93674,0
C00879=48680,52460,-120680,63110,-119873,-93652,0
C00880=48607,52482,-120604,63200,-119875,-93620,0
C00881=48558,52500,-120543,63262,-119880,-93596,0
C00882=48513,52520,-120475,63321,-119890,-93570,0
C00883=48448,52551,-120371,63407,-119905,-93531,0
C00884=48409,52572,-120298,63459,-119919,-93505,0
C00885=48374,52596,-120218,63509,-119936,-93477,0
C00886=48332,52626,-120117,63569,-119958,-93443,0
C00887=48292,52659,-120006,63628,-119986,-93406,0
C00888=48247,52710,-119837,63701,-120032,-93352,0
C00889=48230,52731,-119765,63730,-120052,-93329,0
C00890=48213,52757,-119679,63760,-120079,-93302,0
C00891=48200,52786,-119585,63788,-120109,-93274,0
C00892=48184,52824,-119457,63823,-120150,-93236,0
C00893=48174,52864,-119327,63853,-120195,-93197,0
C00894=48173,52933,-119097,63886,-120280,-93132,0
C00895=48179,52974,-118964,63899,-120332,-93095,0
C00896=48203,53028,-118789,63897,-120406,-93049,0
C00897=48234,53081,-118617,63889,-120482,-93005,0
C00898=48278,53132,-118452,63864,-120560,-92964,0
C00899=48328,53182,-118292,63833,-120638,-92926,0
C00900=48410,53241,-118101,63771,-120742,-92884,0
C00901=48454,53322,-117841,63760,-120854,-92818,0
C00902=39622,59390,-99557,75854,-122076,-86295,0
C00903=39566,59365,-99627,75899,-122025,-86307,0
C00904=39518,59344,-99684,75938,-121984,-86316,0
C00905=39466,59327,-99732,75982,-121941,-86323,0
C00906=39409,59312,-99772,76032,-121898,-86326,0
C00907=39355,59300,-99806,76080,-121858,-86329,0
C00908=39302,59291,-99829,76130,-121821,-86327,0
C00909=39244,59286,-99843,76185,-121784,-86323,0
C00910=39203,59282,-99851,76225,-121758,-86320,0
C00911=39119,59281,-99854,76307,-121707,-86309,0
C00912=39036,59284,-99843,76391,-121661,-86294,0
C00913=38954,59296,-99809,76478,-121621,-86273,0
C00914=38873,59312,-99762,76566,-121584,-86249,0
C00915=38796,59337,-99690,76653,-121555,-86217,0
C00916=38721,59366,-99608,76740,-121530,-86183,0
C00917=38651,59403,-99503,76826,-121514,-86143,0
C00918=38585,59444,-99388,76909,-121501,-86101,0
C00919=38526,59491,-99253,76988,-121498,-86054,0
C00920=38471,59542,-99110,77064,-121498,-86005,0
C00921=38425,59599,-98951,77134,-121507,-85953,0
C00922=38383,59658,-98786,77201,-121521,-85899,0
C00923=38352,59722,-98608,77260,-121543,-85843,0
C00924=38325,59787,-98427,77314,-121569,-85787,0
C00925=38309,59855,-98238,77359,-121602,-85731,0
C00926=38302,59897,-98119,77385,-121625,-85696,0
C00927=38293,59993,-97854,77435,-121681,-85618,0
C00928=38295,60052,-97689,77459,-121720,-85571,0
C00929=38308,60134,-97464,77482,-121778,-85508,0
C00930=38324,60193,-97300,77492,-121825,-85462,0
C00931=38354,60272,-97085,77496,-121893,-85404,0
C00932=38385,60330,-96923,77492,-121950,-85362,0
C00933=38432,60401,-96729,77476,-122022,-85313,0
C00934=38476,60455,-96581,77457,-122083,-85277,0
C00935=38538,60517,-96413,77424,-122160,-85237,0
C00936=38594,60564,-96284,77390,-122224,-85208,0
C00937=38668,60614,-96148,77339,-122301,-85179,0
C00938=38735,60652,-96045,77291,-122367,-85159,0
C00939=38779,60671,-95992,77256,-122406,-85150,0
C00940=38834,60695,-95930,77213,-122454,-85140,0
C00941=38893,60715,-95875,77164,-122503,-85133,0
C00942=38982,60737,-95818,77087,-122572,-85129,0
C00943=39019,60744,-95799,77054,-122600,-85129,0
C00944=39063,60750,-95781,77014,-122631,-85130,0
C00945=39111,60754,-95774,76968,-122663,-85135,0
C00946=39175,60757,-95766,76907,-122705,-85142,0
C00947=39240,60756,-95770,76843,-122745,-85152,0
C00948=39351,60742,-95809,76728,-122805,-85180,0
C00949=39416,60730,-95843,76660,-122837,-85199,0
C00950=39498,60702,-95922,76566,-122869,-85234,0
C00951=39578,60670,-96012,76473,-122898,-85271,0
C00952=39653,60629,-96127,76381,-122917,-85315,0
C00953=39724,60583,-96253,76290,-122931,-85361,0
C00954=39788,60530,-96400,76203,-122936,-85413,0
C00955=39849,60474,-96557,76118,-122936,-85467,0
C00956=39899,60411,-96731,76039,-122925,-85524,0
C00957=39937,60359,-96874,75979,-122914,-85571,0
C00958=39946,60346,-96912,75963,-122910,-85583,0
C00959=39964,60310,-97010,75929,-122898,-85614,0
C00960=39979,60274,-97109,75898,-122883,-85644,0
C00961=40007,60199,-97318,75836,-122849,-85708,0
C00962=40019,60145,-97467,75799,-122821,-85752,0
C00963=40027,60090,-97618,75766,-122788,-85797,0
C00964=40032,60049,-97732,75743,-122764,-85830,0
C00965=40033,60011,-97839,75725,-122739,-85861,0
C00966=40031,59978,-97928,75712,-122716,-85886,0
C00967=40023,59900,-98146,75684,-122657,-85947,0
C00968=40010,59846,-98295,75673,-122614,-85988,0
C00969=39994,59797,-98431,75667,-122571,-86025,0
C00970=39979,59756,-98544,75663,-122534,-86055,0
C00971=39960,59718,-98649,75664,-122498,-86083,0
C00972=39927,59663,-98803,75673,-122440,-86122,0
C00973=39902,59625,-98908,75680,-122400,-86149,0
C00974=39875,59590,-99005,75692,-122360,-86173,0
C00975=39831,59543,-99135,75715,-122302,-86203,0
C00976=39798,59511,-99224,75732,-122261,-86224,0
C00977=39761,59480,-99309,75755,-122218,-86243,0
C00978=39709,59443,-99412,75791,-122162,-86265,0
C00979=39692,59432,-99444,75803,-122145,-86272,0
C00980=39621,59373,-99605,75848,-122063,-86308,0
C00981=29169,52326,-120674,61995,-120075,-93729,0
C00982=29228,52335,-120645,61935,-120109,-93730,0
C00983=29300,52345,-120612,61861,-120148,-93730,0
C00984=29377,52353,-120587,61780,-120186,-93735,0
//INST
///DATE 2025/02/20 16:20
///COMM Generated using RoboDK
///ATTR SC,RW
///GROUP1 RB1
NOP
MOVL C00000 V=60.0 PL=1
MOVL C00001 V=60.0 PL=1
MOVL C00002 V=60.0 PL=1
MOVL C00003 V=60.0 PL=1
MOVL C00004 V=60.0 PL=1
MOVL C00005 V=130.0 PL=1
MOVL C00006 V=60.0 PL=1
MOVL C00007 V=60.0 PL=1
MOVL C00008 V=60.0 PL=1
MOVL C00009 V=60.0 PL=1
MOVL C00010 V=60.0 PL=1
MOVL C00011 V=60.0 PL=1
MOVL C00012 V=60.0 PL=1
MOVL C00013 V=60.0 PL=1
MOVL C00014 V=60.0 PL=1
MOVL C00015 V=60.0 PL=1
MOVL C00016 V=60.0 PL=1
MOVL C00017 V=60.0 PL=1
MOVL C00018 V=60.0 PL=1
MOVL C00019 V=60.0 PL=1
MOVL C00020 V=60.0 PL=1
MOVL C00021 V=60.0 PL=1
MOVL C00022 V=60.0 PL=1
MOVL C00023 V=60.0 PL=1
MOVL C00024 V=60.0 PL=1
MOVL C00025 V=60.0 PL=1
MOVL C00026 V=60.0 PL=1
MOVL C00027 V=60.0 PL=1
MOVL C00028 V=60.0 PL=1
MOVL C00029 V=60.0 PL=1
MOVL C00030 V=60.0 PL=1
MOVL C00031 V=60.0 PL=1
MOVL C00032 V=60.0 PL=1
MOVL C00033 V=60.0 PL=1
MOVL C00034 V=60.0 PL=1
MOVL C00035 V=60.0 PL=1
MOVL C00036 V=60.0 PL=1
MOVL C00037 V=60.0 PL=1
MOVL C00038 V=60.0 PL=1
MOVL C00039 V=60.0 PL=1
MOVL C00040 V=60.0 PL=1
MOVL C00041 V=60.0 PL=1
MOVL C00042 V=60.0 PL=1
MOVL C00043 V=60.0 PL=1
MOVL C00044 V=60.0 PL=1
MOVL C00045 V=60.0 PL=1
MOVL C00046 V=60.0 PL=1
MOVL C00047 V=60.0 PL=1
MOVL C00048 V=130.0 PL=1
MOVL C00049 V=30.0 PL=1
MOVL C00050 V=30.0 PL=1
MOVL C00051 V=30.0 PL=1
MOVL C00052 V=30.0 PL=1
MOVL C00053 V=30.0 PL=1
MOVL C00054 V=30.0 PL=1
MOVL C00055 V=30.0 PL=1
MOVL C00056 V=30.0 PL=1
MOVL C00057 V=30.0 PL=1
MOVL C00058 V=30.0 PL=1
MOVL C00059 V=30.0 PL=1
MOVL C00060 V=30.0 PL=1
MOVL C00061 V=30.0 PL=1
MOVL C00062 V=30.0 PL=1
MOVL C00063 V=30.0 PL=1
MOVL C00064 V=30.0 PL=1
MOVL C00065 V=30.0 PL=1
MOVL C00066 V=30.0 PL=1
MOVL C00067 V=30.0 PL=1
MOVL C00068 V=30.0 PL=1
MOVL C00069 V=30.0 PL=1
MOVL C00070 V=30.0 PL=1
MOVL C00071 V=30.0 PL=1
MOVL C00072 V=30.0 PL=1
MOVL C00073 V=30.0 PL=1
MOVL C00074 V=30.0 PL=1
MOVL C00075 V=30.0 PL=1
MOVL C00076 V=30.0 PL=1
MOVL C00077 V=30.0 PL=1
MOVL C00078 V=30.0 PL=1
MOVL C00079 V=30.0 PL=1
MOVL C00080 V=30.0 PL=1
MOVL C00081 V=30.0 PL=1
MOVL C00082 V=30.0 PL=1
MOVL C00083 V=30.0 PL=1
MOVL C00084 V=30.0 PL=1
MOVL C00085 V=30.0 PL=1
MOVL C00086 V=30.0 PL=1
MOVL C00087 V=30.0 PL=1
MOVL C00088 V=30.0 PL=1
MOVL C00089 V=30.0 PL=1
MOVL C00090 V=30.0 PL=1
MOVL C00091 V=30.0 PL=1
MOVL C00092 V=30.0 PL=1
MOVL C00093 V=30.0 PL=1
MOVL C00094 V=30.0 PL=1
MOVL C00095 V=30.0 PL=1
MOVL C00096 V=30.0 PL=1
MOVL C00097 V=30.0 PL=1
MOVL C00098 V=30.0 PL=1
MOVL C00099 V=30.0 PL=1
MOVL C00100 V=30.0 PL=1
MOVL C00101 V=30.0 PL=1
MOVL C00102 V=30.0 PL=1
MOVL C00103 V=30.0 PL=1
MOVL C00104 V=30.0 PL=1
MOVL C00105 V=30.0 PL=1
MOVL C00106 V=30.0 PL=1
MOVL C00107 V=30.0 PL=1
MOVL C00108 V=30.0 PL=1
MOVL C00109 V=30.0 PL=1
MOVL C00110 V=30.0 PL=1
MOVL C00111 V=30.0 PL=1
MOVL C00112 V=30.0 PL=1
MOVL C00113 V=30.0 PL=1
MOVL C00114 V=30.0 PL=1
MOVL C00115 V=30.0 PL=1
MOVL C00116 V=30.0 PL=1
MOVL C00117 V=30.0 PL=1
MOVL C00118 V=30.0 PL=1
MOVL C00119 V=30.0 PL=1
MOVL C00120 V=30.0 PL=1
MOVL C00121 V=130.0 PL=1
MOVL C00122 V=130.0 PL=1
MOVL C00123 V=30.0 PL=1
MOVL C00124 V=30.0 PL=1
MOVL C00125 V=30.0 PL=1
MOVL C00126 V=30.0 PL=1
MOVL C00127 V=30.0 PL=1
MOVL C00128 V=30.0 PL=1
MOVL C00129 V=30.0 PL=1
MOVL C00130 V=30.0 PL=1
MOVL C00131 V=30.0 PL=1
MOVL C00132 V=30.0 PL=1
MOVL C00133 V=30.0 PL=1
MOVL C00134 V=30.0 PL=1
MOVL C00135 V=30.0 PL=1
MOVL C00136 V=30.0 PL=1
MOVL C00137 V=30.0 PL=1
MOVL C00138 V=30.0 PL=1
MOVL C00139 V=30.0 PL=1
MOVL C00140 V=30.0 PL=1
MOVL C00141 V=30.0 PL=1
MOVL C00142 V=30.0 PL=1
MOVL C00143 V=30.0 PL=1
MOVL C00144 V=30.0 PL=1
MOVL C00145 V=30.0 PL=1
MOVL C00146 V=30.0 PL=1
MOVL C00147 V=30.0 PL=1
MOVL C00148 V=30.0 PL=1
MOVL C00149 V=30.0 PL=1
MOVL C00150 V=30.0 PL=1
MOVL C00151 V=30.0 PL=1
MOVL C00152 V=30.0 PL=1
MOVL C00153 V=30.0 PL=1
MOVL C00154 V=30.0 PL=1
MOVL C00155 V=30.0 PL=1
MOVL C00156 V=30.0 PL=1
MOVL C00157 V=30.0 PL=1
MOVL C00158 V=30.0 PL=1
MOVL C00159 V=30.0 PL=1
MOVL C00160 V=30.0 PL=1
MOVL C00161 V=30.0 PL=1
MOVL C00162 V=30.0 PL=1
MOVL C00163 V=30.0 PL=1
MOVL C00164 V=30.0 PL=1
MOVL C00165 V=30.0 PL=1
MOVL C00166 V=30.0 PL=1
MOVL C00167 V=30.0 PL=1
MOVL C00168 V=30.0 PL=1
MOVL C00169 V=30.0 PL=1
MOVL C00170 V=30.0 PL=1
MOVL C00171 V=30.0 PL=1
MOVL C00172 V=30.0 PL=1
MOVL C00173 V=30.0 PL=1
MOVL C00174 V=30.0 PL=1
MOVL C00175 V=30.0 PL=1
MOVL C00176 V=30.0 PL=1
MOVL C00177 V=30.0 PL=1
MOVL C00178 V=30.0 PL=1
MOVL C00179 V=30.0 PL=1
MOVL C00180 V=30.0 PL=1
MOVL C00181 V=30.0 PL=1
MOVL C00182 V=30.0 PL=1
MOVL C00183 V=30.0 PL=1
MOVL C00184 V=30.0 PL=1
MOVL C00185 V=30.0 PL=1
MOVL C00186 V=30.0 PL=1
MOVL C00187 V=30.0 PL=1
MOVL C00188 V=30.0 PL=1
MOVL C00189 V=30.0 PL=1
MOVL C00190 V=30.0 PL=1
MOVL C00191 V=30.0 PL=1
MOVL C00192 V=30.0 PL=1
MOVL C00193 V=30.0 PL=1
MOVL C00194 V=30.0 PL=1
MOVL C00195 V=30.0 PL=1
MOVL C00196 V=30.0 PL=1
MOVL C00197 V=30.0 PL=1
MOVL C00198 V=30.0 PL=1
MOVL C00199 V=30.0 PL=1
MOVL C00200 V=30.0 PL=1
MOVL C00201 V=30.0 PL=1
MOVL C00202 V=30.0 PL=1
MOVL C00203 V=30.0 PL=1
MOVL C00204 V=30.0 PL=1
MOVL C00205 V=30.0 PL=1
MOVL C00206 V=30.0 PL=1
MOVL C00207 V=30.0 PL=1
MOVL C00208 V=30.0 PL=1
MOVL C00209 V=30.0 PL=1
MOVL C00210 V=30.0 PL=1
MOVL C00211 V=30.0 PL=1
MOVL C00212 V=30.0 PL=1
MOVL C00213 V=30.0 PL=1
MOVL C00214 V=130.0 PL=1
MOVL C00215 V=30.0 PL=1
MOVL C00216 V=30.0 PL=1
MOVL C00217 V=30.0 PL=1
MOVL C00218 V=30.0 PL=1
MOVL C00219 V=30.0 PL=1
MOVL C00220 V=30.0 PL=1
MOVL C00221 V=30.0 PL=1
MOVL C00222 V=30.0 PL=1
MOVL C00223 V=30.0 PL=1
MOVL C00224 V=30.0 PL=1
MOVL C00225 V=30.0 PL=1
MOVL C00226 V=30.0 PL=1
MOVL C00227 V=30.0 PL=1
MOVL C00228 V=30.0 PL=1
MOVL C00229 V=30.0 PL=1
MOVL C00230 V=30.0 PL=1
MOVL C00231 V=30.0 PL=1
MOVL C00232 V=30.0 PL=1
MOVL C00233 V=30.0 PL=1
MOVL C00234 V=30.0 PL=1
MOVL C00235 V=30.0 PL=1
MOVL C00236 V=30.0 PL=1
MOVL C00237 V=30.0 PL=1
MOVL C00238 V=30.0 PL=1
MOVL C00239 V=30.0 PL=1
MOVL C00240 V=30.0 PL=1
MOVL C00241 V=30.0 PL=1
MOVL C00242 V=30.0 PL=1
MOVL C00243 V=30.0 PL=1
MOVL C00244 V=30.0 PL=1
MOVL C00245 V=30.0 PL=1
MOVL C00246 V=30.0 PL=1
MOVL C00247 V=30.0 PL=1
MOVL C00248 V=30.0 PL=1
MOVL C00249 V=30.0 PL=1
MOVL C00250 V=30.0 PL=1
MOVL C00251 V=30.0 PL=1
MOVL C00252 V=30.0 PL=1
MOVL C00253 V=30.0 PL=1
MOVL C00254 V=30.0 PL=1
MOVL C00255 V=30.0 PL=1
MOVL C00256 V=30.0 PL=1
MOVL C00257 V=30.0 PL=1
MOVL C00258 V=30.0 PL=1
MOVL C00259 V=30.0 PL=1
MOVL C00260 V=30.0 PL=1
MOVL C00261 V=30.0 PL=1
MOVL C00262 V=30.0 PL=1
MOVL C00263 V=30.0 PL=1
MOVL C00264 V=30.0 PL=1
MOVL C00265 V=30.0 PL=1
MOVL C00266 V=30.0 PL=1
MOVL C00267 V=30.0 PL=1
MOVL C00268 V=30.0 PL=1
MOVL C00269 V=30.0 PL=1
MOVL C00270 V=30.0 PL=1
MOVL C00271 V=30.0 PL=1
MOVL C00272 V=30.0 PL=1
MOVL C00273 V=30.0 PL=1
MOVL C00274 V=30.0 PL=1
MOVL C00275 V=30.0 PL=1
MOVL C00276 V=30.0 PL=1
MOVL C00277 V=30.0 PL=1
MOVL C00278 V=30.0 PL=1
MOVL C00279 V=30.0 PL=1
MOVL C00280 V=30.0 PL=1
MOVL C00281 V=30.0 PL=1
MOVL C00282 V=30.0 PL=1
MOVL C00283 V=30.0 PL=1
MOVL C00284 V=30.0 PL=1
MOVL C00285 V=30.0 PL=1
MOVL C00286 V=30.0 PL=1
MOVL C00287 V=30.0 PL=1
MOVL C00288 V=30.0 PL=1
MOVL C00289 V=30.0 PL=1
MOVL C00290 V=30.0 PL=1
MOVL C00291 V=30.0 PL=1
MOVL C00292 V=30.0 PL=1
MOVL C00293 V=30.0 PL=1
MOVL C00294 V=30.0 PL=1
MOVL C00295 V=30.0 PL=1
MOVL C00296 V=30.0 PL=1
MOVL C00297 V=30.0 PL=1
MOVL C00298 V=30.0 PL=1
MOVL C00299 V=30.0 PL=1
MOVL C00300 V=30.0 PL=1
MOVL C00301 V=30.0 PL=1
MOVL C00302 V=30.0 PL=1
MOVL C00303 V=30.0 PL=1
MOVL C00304 V=130.0 PL=1
MOVL C00305 V=15.0 PL=1
MOVL C00306 V=15.0 PL=1
MOVL C00307 V=15.0 PL=1
MOVL C00308 V=15.0 PL=1
MOVL C00309 V=15.0 PL=1
MOVL C00310 V=15.0 PL=1
MOVL C00311 V=15.0 PL=1
MOVL C00312 V=15.0 PL=1
MOVL C00313 V=15.0 PL=1
MOVL C00314 V=15.0 PL=1
MOVL C00315 V=15.0 PL=1
MOVL C00316 V=15.0 PL=1
MOVL C00317 V=15.0 PL=1
MOVL C00318 V=15.0 PL=1
MOVL C00319 V=15.0 PL=1
MOVL C00320 V=15.0 PL=1
MOVL C00321 V=15.0 PL=1
MOVL C00322 V=15.0 PL=1
MOVL C00323 V=15.0 PL=1
MOVL C00324 V=15.0 PL=1
MOVL C00325 V=15.0 PL=1
MOVL C00326 V=15.0 PL=1
MOVL C00327 V=15.0 PL=1
MOVL C00328 V=15.0 PL=1
MOVL C00329 V=130.0 PL=1
MOVL C00330 V=15.0 PL=1
MOVL C00331 V=130.0 PL=1
MOVL C00332 V=15.0 PL=1
MOVL C00333 V=15.0 PL=1
MOVL C00334 V=15.0 PL=1
MOVL C00335 V=15.0 PL=1
MOVL C00336 V=15.0 PL=1
MOVL C00337 V=15.0 PL=1
MOVL C00338 V=15.0 PL=1
MOVL C00339 V=15.0 PL=1
MOVL C00340 V=15.0 PL=1
MOVL C00341 V=15.0 PL=1
MOVL C00342 V=15.0 PL=1
MOVL C00343 V=15.0 PL=1
MOVL C00344 V=15.0 PL=1
MOVL C00345 V=15.0 PL=1
MOVL C00346 V=15.0 PL=1
MOVL C00347 V=15.0 PL=1
MOVL C00348 V=15.0 PL=1
MOVL C00349 V=15.0 PL=1
MOVL C00350 V=15.0 PL=1
MOVL C00351 V=15.0 PL=1
MOVL C00352 V=15.0 PL=1
MOVL C00353 V=15.0 PL=1
MOVL C00354 V=15.0 PL=1
MOVL C00355 V=15.0 PL=1
MOVL C00356 V=15.0 PL=1
MOVL C00357 V=15.0 PL=1
MOVL C00358 V=15.0 PL=1
MOVL C00359 V=15.0 PL=1
MOVL C00360 V=15.0 PL=1
MOVL C00361 V=15.0 PL=1
MOVL C00362 V=15.0 PL=1
MOVL C00363 V=15.0 PL=1
MOVL C00364 V=15.0 PL=1
MOVL C00365 V=15.0 PL=1
MOVL C00366 V=15.0 PL=1
MOVL C00367 V=15.0 PL=1
MOVL C00368 V=15.0 PL=1
MOVL C00369 V=15.0 PL=1
MOVL C00370 V=15.0 PL=1
MOVL C00371 V=15.0 PL=1
MOVL C00372 V=15.0 PL=1
MOVL C00373 V=15.0 PL=1
MOVL C00374 V=15.0 PL=1
MOVL C00375 V=130.0 PL=1
MOVL C00376 V=80.0 PL=1
MOVL C00377 V=130.0 PL=1
MOVL C00378 V=80.0 PL=1
MOVL C00379 V=80.0 PL=1
MOVL C00380 V=80.0 PL=1
MOVL C00381 V=80.0 PL=1
MOVL C00382 V=130.0 PL=1
MOVL C00383 V=130.0 PL=1
MOVL C00384 V=30.0 PL=1
MOVL C00385 V=30.0 PL=1
MOVL C00386 V=30.0 PL=1
MOVL C00387 V=30.0 PL=1
MOVL C00388 V=30.0 PL=1
MOVL C00389 V=30.0 PL=1
MOVL C00390 V=30.0 PL=1
MOVL C00391 V=30.0 PL=1
MOVL C00392 V=30.0 PL=1
MOVL C00393 V=30.0 PL=1
MOVL C00394 V=30.0 PL=1
MOVL C00395 V=30.0 PL=1
MOVL C00396 V=30.0 PL=1
MOVL C00397 V=30.0 PL=1
MOVL C00398 V=30.0 PL=1
MOVL C00399 V=30.0 PL=1
MOVL C00400 V=30.0 PL=1
MOVL C00401 V=30.0 PL=1
MOVL C00402 V=30.0 PL=1
MOVL C00403 V=30.0 PL=1
MOVL C00404 V=30.0 PL=1
MOVL C00405 V=30.0 PL=1
MOVL C00406 V=30.0 PL=1
MOVL C00407 V=30.0 PL=1
MOVL C00408 V=30.0 PL=1
MOVL C00409 V=30.0 PL=1
MOVL C00410 V=30.0 PL=1
MOVL C00411 V=30.0 PL=1
MOVL C00412 V=30.0 PL=1
MOVL C00413 V=30.0 PL=1
MOVL C00414 V=30.0 PL=1
MOVL C00415 V=30.0 PL=1
MOVL C00416 V=30.0 PL=1
MOVL C00417 V=30.0 PL=1
MOVL C00418 V=30.0 PL=1
MOVL C00419 V=30.0 PL=1
MOVL C00420 V=30.0 PL=1
MOVL C00421 V=30.0 PL=1
MOVL C00422 V=30.0 PL=1
MOVL C00423 V=30.0 PL=1
MOVL C00424 V=30.0 PL=1
MOVL C00425 V=30.0 PL=1
MOVL C00426 V=30.0 PL=1
MOVL C00427 V=30.0 PL=1
MOVL C00428 V=30.0 PL=1
MOVL C00429 V=30.0 PL=1
MOVL C00430 V=30.0 PL=1
MOVL C00431 V=30.0 PL=1
MOVL C00432 V=30.0 PL=1
MOVL C00433 V=30.0 PL=1
MOVL C00434 V=30.0 PL=1
MOVL C00435 V=30.0 PL=1
MOVL C00436 V=30.0 PL=1
MOVL C00437 V=30.0 PL=1
MOVL C00438 V=30.0 PL=1
MOVL C00439 V=30.0 PL=1
MOVL C00440 V=30.0 PL=1
MOVL C00441 V=30.0 PL=1
MOVL C00442 V=30.0 PL=1
MOVL C00443 V=30.0 PL=1
MOVL C00444 V=30.0 PL=1
MOVL C00445 V=30.0 PL=1
MOVL C00446 V=30.0 PL=1
MOVL C00447 V=30.0 PL=1
MOVL C00448 V=30.0 PL=1
MOVL C00449 V=30.0 PL=1
MOVL C00450 V=30.0 PL=1
MOVL C00451 V=30.0 PL=1
MOVL C00452 V=30.0 PL=1
MOVL C00453 V=30.0 PL=1
MOVL C00454 V=30.0 PL=1
MOVL C00455 V=30.0 PL=1
MOVL C00456 V=30.0 PL=1
MOVL C00457 V=30.0 PL=1
MOVL C00458 V=30.0 PL=1
MOVL C00459 V=30.0 PL=1
MOVL C00460 V=130.0 PL=1
MOVL C00461 V=130.0 PL=1
MOVL C00462 V=60.0 PL=1
MOVL C00463 V=60.0 PL=1
MOVL C00464 V=60.0 PL=1
MOVL C00465 V=60.0 PL=1
MOVL C00466 V=130.0 PL=1
MOVL C00467 V=30.0 PL=1
MOVL C00468 V=30.0 PL=1
MOVL C00469 V=30.0 PL=1
MOVL C00470 V=30.0 PL=1
MOVL C00471 V=30.0 PL=1
MOVL C00472 V=30.0 PL=1
MOVL C00473 V=30.0 PL=1
MOVL C00474 V=30.0 PL=1
MOVL C00475 V=130.0 PL=1
MOVL C00476 V=130.0 PL=1
MOVL C00477 V=30.0 PL=1
MOVL C00478 V=130.0 PL=1
MOVL C00479 V=30.0 PL=1
MOVL C00480 V=130.0 PL=1
MOVL C00481 V=30.0 PL=1
MOVL C00482 V=130.0 PL=1
MOVL C00483 V=20.0 PL=1
MOVL C00484 V=130.0 PL=1
MOVL C00485 V=30.0 PL=1
MOVL C00486 V=30.0 PL=1
MOVL C00487 V=30.0 PL=1
MOVL C00488 V=30.0 PL=1
MOVL C00489 V=30.0 PL=1
MOVL C00490 V=30.0 PL=1
MOVL C00491 V=30.0 PL=1
MOVL C00492 V=30.0 PL=1
MOVL C00493 V=30.0 PL=1
MOVL C00494 V=30.0 PL=1
MOVL C00495 V=30.0 PL=1
MOVL C00496 V=30.0 PL=1
MOVL C00497 V=30.0 PL=1
MOVL C00498 V=30.0 PL=1
MOVL C00499 V=30.0 PL=1
MOVL C00500 V=30.0 PL=1
MOVL C00501 V=30.0 PL=1
MOVL C00502 V=30.0 PL=1
MOVL C00503 V=30.0 PL=1
MOVL C00504 V=30.0 PL=1
MOVL C00505 V=30.0 PL=1
MOVL C00506 V=30.0 PL=1
MOVL C00507 V=30.0 PL=1
MOVL C00508 V=30.0 PL=1
MOVL C00509 V=30.0 PL=1
MOVL C00510 V=30.0 PL=1
MOVL C00511 V=30.0 PL=1
MOVL C00512 V=30.0 PL=1
MOVL C00513 V=30.0 PL=1
MOVL C00514 V=30.0 PL=1
MOVL C00515 V=30.0 PL=1
MOVL C00516 V=30.0 PL=1
MOVL C00517 V=30.0 PL=1
MOVL C00518 V=30.0 PL=1
MOVL C00519 V=30.0 PL=1
MOVL C00520 V=30.0 PL=1
MOVL C00521 V=30.0 PL=1
MOVL C00522 V=30.0 PL=1
MOVL C00523 V=30.0 PL=1
MOVL C00524 V=30.0 PL=1
MOVL C00525 V=30.0 PL=1
MOVL C00526 V=30.0 PL=1
MOVL C00527 V=30.0 PL=1
MOVL C00528 V=30.0 PL=1
MOVL C00529 V=30.0 PL=1
MOVL C00530 V=30.0 PL=1
MOVL C00531 V=30.0 PL=1
MOVL C00532 V=30.0 PL=1
MOVL C00533 V=30.0 PL=1
MOVL C00534 V=30.0 PL=1
MOVL C00535 V=30.0 PL=1
MOVL C00536 V=30.0 PL=1
MOVL C00537 V=30.0 PL=1
MOVL C00538 V=30.0 PL=1
MOVL C00539 V=30.0 PL=1
MOVL C00540 V=30.0 PL=1
MOVL C00541 V=30.0 PL=1
MOVL C00542 V=30.0 PL=1
MOVL C00543 V=30.0 PL=1
MOVL C00544 V=30.0 PL=1
MOVL C00545 V=30.0 PL=1
MOVL C00546 V=30.0 PL=1
MOVL C00547 V=30.0 PL=1
MOVL C00548 V=30.0 PL=1
MOVL C00549 V=30.0 PL=1
MOVL C00550 V=30.0 PL=1
MOVL C00551 V=30.0 PL=1
MOVL C00552 V=30.0 PL=1
MOVL C00553 V=30.0 PL=1
MOVL C00554 V=30.0 PL=1
MOVL C00555 V=30.0 PL=1
MOVL C00556 V=30.0 PL=1
MOVL C00557 V=30.0 PL=1
MOVL C00558 V=30.0 PL=1
MOVL C00559 V=30.0 PL=1
MOVL C00560 V=30.0 PL=1
MOVL C00561 V=130.0 PL=1
MOVL C00562 V=130.0 PL=1
MOVL C00563 V=30.0 PL=1
MOVL C00564 V=30.0 PL=1
MOVL C00565 V=30.0 PL=1
MOVL C00566 V=30.0 PL=1
MOVL C00567 V=30.0 PL=1
MOVL C00568 V=30.0 PL=1
MOVL C00569 V=30.0 PL=1
MOVL C00570 V=30.0 PL=1
MOVL C00571 V=30.0 PL=1
MOVL C00572 V=30.0 PL=1
MOVL C00573 V=30.0 PL=1
MOVL C00574 V=30.0 PL=1
MOVL C00575 V=30.0 PL=1
MOVL C00576 V=30.0 PL=1
MOVL C00577 V=30.0 PL=1
MOVL C00578 V=30.0 PL=1
MOVL C00579 V=30.0 PL=1
MOVL C00580 V=30.0 PL=1
MOVL C00581 V=30.0 PL=1
MOVL C00582 V=30.0 PL=1
MOVL C00583 V=30.0 PL=1
MOVL C00584 V=30.0 PL=1
MOVL C00585 V=30.0 PL=1
MOVL C00586 V=30.0 PL=1
MOVL C00587 V=30.0 PL=1
MOVL C00588 V=30.0 PL=1
MOVL C00589 V=30.0 PL=1
MOVL C00590 V=30.0 PL=1
MOVL C00591 V=30.0 PL=1
MOVL C00592 V=30.0 PL=1
MOVL C00593 V=30.0 PL=1
MOVL C00594 V=30.0 PL=1
MOVL C00595 V=30.0 PL=1
MOVL C00596 V=30.0 PL=1
MOVL C00597 V=30.0 PL=1
MOVL C00598 V=30.0 PL=1
MOVL C00599 V=30.0 PL=1
MOVL C00600 V=30.0 PL=1
MOVL C00601 V=30.0 PL=1
MOVL C00602 V=30.0 PL=1
MOVL C00603 V=30.0 PL=1
MOVL C00604 V=30.0 PL=1
MOVL C00605 V=30.0 PL=1
MOVL C00606 V=30.0 PL=1
MOVL C00607 V=30.0 PL=1
MOVL C00608 V=30.0 PL=1
MOVL C00609 V=30.0 PL=1
MOVL C00610 V=30.0 PL=1
MOVL C00611 V=30.0 PL=1
MOVL C00612 V=30.0 PL=1
MOVL C00613 V=30.0 PL=1
MOVL C00614 V=30.0 PL=1
MOVL C00615 V=30.0 PL=1
MOVL C00616 V=30.0 PL=1
MOVL C00617 V=30.0 PL=1
MOVL C00618 V=30.0 PL=1
MOVL C00619 V=30.0 PL=1
MOVL C00620 V=30.0 PL=1
MOVL C00621 V=30.0 PL=1
MOVL C00622 V=30.0 PL=1
MOVL C00623 V=30.0 PL=1
MOVL C00624 V=30.0 PL=1
MOVL C00625 V=30.0 PL=1
MOVL C00626 V=30.0 PL=1
MOVL C00627 V=30.0 PL=1
MOVL C00628 V=30.0 PL=1
MOVL C00629 V=30.0 PL=1
MOVL C00630 V=30.0 PL=1
MOVL C00631 V=30.0 PL=1
MOVL C00632 V=30.0 PL=1
MOVL C00633 V=30.0 PL=1
MOVL C00634 V=30.0 PL=1
MOVL C00635 V=30.0 PL=1
MOVL C00636 V=30.0 PL=1
MOVL C00637 V=130.0 PL=1
MOVL C00638 V=130.0 PL=1
MOVL C00639 V=30.0 PL=1
MOVL C00640 V=130.0 PL=1
MOVL C00641 V=30.0 PL=1
MOVL C00642 V=30.0 PL=1
MOVL C00643 V=30.0 PL=1
MOVL C00644 V=30.0 PL=1
MOVL C00645 V=30.0 PL=1
MOVL C00646 V=30.0 PL=1
MOVL C00647 V=30.0 PL=1
MOVL C00648 V=30.0 PL=1
MOVL C00649 V=30.0 PL=1
MOVL C00650 V=30.0 PL=1
MOVL C00651 V=30.0 PL=1
MOVL C00652 V=30.0 PL=1
MOVL C00653 V=30.0 PL=1
MOVL C00654 V=30.0 PL=1
MOVL C00655 V=30.0 PL=1
MOVL C00656 V=30.0 PL=1
MOVL C00657 V=30.0 PL=1
MOVL C00658 V=30.0 PL=1
MOVL C00659 V=30.0 PL=1
MOVL C00660 V=30.0 PL=1
MOVL C00661 V=30.0 PL=1
MOVL C00662 V=30.0 PL=1
MOVL C00663 V=30.0 PL=1
MOVL C00664 V=30.0 PL=1
MOVL C00665 V=30.0 PL=1
MOVL C00666 V=30.0 PL=1
MOVL C00667 V=30.0 PL=1
MOVL C00668 V=30.0 PL=1
MOVL C00669 V=30.0 PL=1
MOVL C00670 V=30.0 PL=1
MOVL C00671 V=30.0 PL=1
MOVL C00672 V=30.0 PL=1
MOVL C00673 V=30.0 PL=1
MOVL C00674 V=30.0 PL=1
MOVL C00675 V=30.0 PL=1
MOVL C00676 V=30.0 PL=1
MOVL C00677 V=30.0 PL=1
MOVL C00678 V=30.0 PL=1
MOVL C00679 V=30.0 PL=1
MOVL C00680 V=30.0 PL=1
MOVL C00681 V=30.0 PL=1
MOVL C00682 V=30.0 PL=1
MOVL C00683 V=30.0 PL=1
MOVL C00684 V=30.0 PL=1
MOVL C00685 V=30.0 PL=1
MOVL C00686 V=30.0 PL=1
MOVL C00687 V=30.0 PL=1
MOVL C00688 V=30.0 PL=1
MOVL C00689 V=30.0 PL=1
MOVL C00690 V=30.0 PL=1
MOVL C00691 V=30.0 PL=1
MOVL C00692 V=30.0 PL=1
MOVL C00693 V=30.0 PL=1
MOVL C00694 V=30.0 PL=1
MOVL C00695 V=30.0 PL=1
MOVL C00696 V=30.0 PL=1
MOVL C00697 V=30.0 PL=1
MOVL C00698 V=30.0 PL=1
MOVL C00699 V=30.0 PL=1
MOVL C00700 V=30.0 PL=1
MOVL C00701 V=30.0 PL=1
MOVL C00702 V=30.0 PL=1
MOVL C00703 V=30.0 PL=1
MOVL C00704 V=30.0 PL=1
MOVL C00705 V=30.0 PL=1
MOVL C00706 V=30.0 PL=1
MOVL C00707 V=30.0 PL=1
MOVL C00708 V=30.0 PL=1
MOVL C00709 V=30.0 PL=1
MOVL C00710 V=30.0 PL=1
MOVL C00711 V=30.0 PL=1
MOVL C00712 V=30.0 PL=1
MOVL C00713 V=30.0 PL=1
MOVL C00714 V=30.0 PL=1
MOVL C00715 V=130.0 PL=1
MOVL C00716 V=130.0 PL=1
MOVL C00717 V=130.0 PL=1
MOVL C00718 V=30.0 PL=1
MOVL C00719 V=30.0 PL=1
MOVL C00720 V=30.0 PL=1
MOVL C00721 V=30.0 PL=1
MOVL C00722 V=30.0 PL=1
MOVL C00723 V=30.0 PL=1
MOVL C00724 V=30.0 PL=1
MOVL C00725 V=30.0 PL=1
MOVL C00726 V=30.0 PL=1
MOVL C00727 V=30.0 PL=1
MOVL C00728 V=30.0 PL=1
MOVL C00729 V=30.0 PL=1
MOVL C00730 V=30.0 PL=1
MOVL C00731 V=30.0 PL=1
MOVL C00732 V=30.0 PL=1
MOVL C00733 V=30.0 PL=1
MOVL C00734 V=30.0 PL=1
MOVL C00735 V=30.0 PL=1
MOVL C00736 V=30.0 PL=1
MOVL C00737 V=30.0 PL=1
MOVL C00738 V=30.0 PL=1
MOVL C00739 V=30.0 PL=1
MOVL C00740 V=30.0 PL=1
MOVL C00741 V=30.0 PL=1
MOVL C00742 V=30.0 PL=1
MOVL C00743 V=30.0 PL=1
MOVL C00744 V=30.0 PL=1
MOVL C00745 V=30.0 PL=1
MOVL C00746 V=30.0 PL=1
MOVL C00747 V=30.0 PL=1
MOVL C00748 V=30.0 PL=1
MOVL C00749 V=30.0 PL=1
MOVL C00750 V=30.0 PL=1
MOVL C00751 V=30.0 PL=1
MOVL C00752 V=30.0 PL=1
MOVL C00753 V=30.0 PL=1
MOVL C00754 V=30.0 PL=1
MOVL C00755 V=30.0 PL=1
MOVL C00756 V=30.0 PL=1
MOVL C00757 V=30.0 PL=1
MOVL C00758 V=30.0 PL=1
MOVL C00759 V=30.0 PL=1
MOVL C00760 V=30.0 PL=1
MOVL C00761 V=30.0 PL=1
MOVL C00762 V=30.0 PL=1
MOVL C00763 V=30.0 PL=1
MOVL C00764 V=30.0 PL=1
MOVL C00765 V=30.0 PL=1
MOVL C00766 V=30.0 PL=1
MOVL C00767 V=30.0 PL=1
MOVL C00768 V=30.0 PL=1
MOVL C00769 V=30.0 PL=1
MOVL C00770 V=30.0 PL=1
MOVL C00771 V=30.0 PL=1
MOVL C00772 V=30.0 PL=1
MOVL C00773 V=30.0 PL=1
MOVL C00774 V=30.0 PL=1
MOVL C00775 V=30.0 PL=1
MOVL C00776 V=30.0 PL=1
MOVL C00777 V=30.0 PL=1
MOVL C00778 V=30.0 PL=1
MOVL C00779 V=30.0 PL=1
MOVL C00780 V=30.0 PL=1
MOVL C00781 V=30.0 PL=1
MOVL C00782 V=30.0 PL=1
MOVL C00783 V=30.0 PL=1
MOVL C00784 V=30.0 PL=1
MOVL C00785 V=30.0 PL=1
MOVL C00786 V=30.0 PL=1
MOVL C00787 V=30.0 PL=1
MOVL C00788 V=30.0 PL=1
MOVL C00789 V=30.0 PL=1
MOVL C00790 V=30.0 PL=1
MOVL C00791 V=30.0 PL=1
MOVL C00792 V=30.0 PL=1
MOVL C00793 V=30.0 PL=1
MOVL C00794 V=30.0 PL=1
MOVL C00795 V=30.0 PL=1
MOVL C00796 V=30.0 PL=1
MOVL C00797 V=30.0 PL=1
MOVL C00798 V=30.0 PL=1
MOVL C00799 V=130.0 PL=1
MOVL C00800 V=130.0 PL=1
MOVL C00801 V=60.0 PL=1
MOVL C00802 V=60.0 PL=1
MOVL C00803 V=60.0 PL=1
MOVL C00804 V=60.0 PL=1
MOVL C00805 V=130.0 PL=1
MOVL C00806 V=30.0 PL=1
MOVL C00807 V=30.0 PL=1
MOVL C00808 V=30.0 PL=1
MOVL C00809 V=30.0 PL=1
MOVL C00810 V=30.0 PL=1
MOVL C00811 V=30.0 PL=1
MOVL C00812 V=30.0 PL=1
MOVL C00813 V=30.0 PL=1
MOVL C00814 V=130.0 PL=1
MOVL C00815 V=130.0 PL=1
MOVL C00816 V=30.0 PL=1
MOVL C00817 V=130.0 PL=1
MOVL C00818 V=30.0 PL=1
MOVL C00819 V=130.0 PL=1
MOVL C00820 V=30.0 PL=1
MOVL C00821 V=130.0 PL=1
MOVL C00822 V=20.0 PL=1
MOVL C00823 V=130.0 PL=1
MOVL C00824 V=30.0 PL=1
MOVL C00825 V=30.0 PL=1
MOVL C00826 V=30.0 PL=1
MOVL C00827 V=30.0 PL=1
MOVL C00828 V=30.0 PL=1
MOVL C00829 V=30.0 PL=1
MOVL C00830 V=30.0 PL=1
MOVL C00831 V=30.0 PL=1
MOVL C00832 V=30.0 PL=1
MOVL C00833 V=30.0 PL=1
MOVL C00834 V=30.0 PL=1
MOVL C00835 V=30.0 PL=1
MOVL C00836 V=30.0 PL=1
MOVL C00837 V=30.0 PL=1
MOVL C00838 V=30.0 PL=1
MOVL C00839 V=30.0 PL=1
MOVL C00840 V=30.0 PL=1
MOVL C00841 V=30.0 PL=1
MOVL C00842 V=30.0 PL=1
MOVL C00843 V=30.0 PL=1
MOVL C00844 V=30.0 PL=1
MOVL C00845 V=30.0 PL=1
MOVL C00846 V=30.0 PL=1
MOVL C00847 V=30.0 PL=1
MOVL C00848 V=30.0 PL=1
MOVL C00849 V=30.0 PL=1
MOVL C00850 V=30.0 PL=1
MOVL C00851 V=30.0 PL=1
MOVL C00852 V=30.0 PL=1
MOVL C00853 V=30.0 PL=1
MOVL C00854 V=30.0 PL=1
MOVL C00855 V=30.0 PL=1
MOVL C00856 V=30.0 PL=1
MOVL C00857 V=30.0 PL=1
MOVL C00858 V=30.0 PL=1
MOVL C00859 V=30.0 PL=1
MOVL C00860 V=30.0 PL=1
MOVL C00861 V=30.0 PL=1
MOVL C00862 V=30.0 PL=1
MOVL C00863 V=30.0 PL=1
MOVL C00864 V=30.0 PL=1
MOVL C00865 V=30.0 PL=1
MOVL C00866 V=30.0 PL=1
MOVL C00867 V=30.0 PL=1
MOVL C00868 V=30.0 PL=1
MOVL C00869 V=30.0 PL=1
MOVL C00870 V=30.0 PL=1
MOVL C00871 V=30.0 PL=1
MOVL C00872 V=30.0 PL=1
MOVL C00873 V=30.0 PL=1
MOVL C00874 V=30.0 PL=1
MOVL C00875 V=30.0 PL=1
MOVL C00876 V=30.0 PL=1
MOVL C00877 V=30.0 PL=1
MOVL C00878 V=30.0 PL=1
MOVL C00879 V=30.0 PL=1
MOVL C00880 V=30.0 PL=1
MOVL C00881 V=30.0 PL=1
MOVL C00882 V=30.0 PL=1
MOVL C00883 V=30.0 PL=1
MOVL C00884 V=30.0 PL=1
MOVL C00885 V=30.0 PL=1
MOVL C00886 V=30.0 PL=1
MOVL C00887 V=30.0 PL=1
MOVL C00888 V=30.0 PL=1
MOVL C00889 V=30.0 PL=1
MOVL C00890 V=30.0 PL=1
MOVL C00891 V=30.0 PL=1
MOVL C00892 V=30.0 PL=1
MOVL C00893 V=30.0 PL=1
MOVL C00894 V=30.0 PL=1
MOVL C00895 V=30.0 PL=1
MOVL C00896 V=30.0 PL=1
MOVL C00897 V=30.0 PL=1
MOVL C00898 V=30.0 PL=1
MOVL C00899 V=30.0 PL=1
MOVL C00900 V=30.0 PL=1
MOVL C00901 V=130.0 PL=1
MOVL C00902 V=130.0 PL=1
MOVL C00903 V=30.0 PL=1
MOVL C00904 V=30.0 PL=1
MOVL C00905 V=30.0 PL=1
MOVL C00906 V=30.0 PL=1
MOVL C00907 V=30.0 PL=1
MOVL C00908 V=30.0 PL=1
MOVL C00909 V=30.0 PL=1
MOVL C00910 V=30.0 PL=1
MOVL C00911 V=30.0 PL=1
MOVL C00912 V=30.0 PL=1
MOVL C00913 V=30.0 PL=1
MOVL C00914 V=30.0 PL=1
MOVL C00915 V=30.0 PL=1
MOVL C00916 V=30.0 PL=1
MOVL C00917 V=30.0 PL=1
MOVL C00918 V=30.0 PL=1
MOVL C00919 V=30.0 PL=1
MOVL C00920 V=30.0 PL=1
MOVL C00921 V=30.0 PL=1
MOVL C00922 V=30.0 PL=1
MOVL C00923 V=30.0 PL=1
MOVL C00924 V=30.0 PL=1
MOVL C00925 V=30.0 PL=1
MOVL C00926 V=30.0 PL=1
MOVL C00927 V=30.0 PL=1
MOVL C00928 V=30.0 PL=1
MOVL C00929 V=30.0 PL=1
MOVL C00930 V=30.0 PL=1
MOVL C00931 V=30.0 PL=1
MOVL C00932 V=30.0 PL=1
MOVL C00933 V=30.0 PL=1
MOVL C00934 V=30.0 PL=1
MOVL C00935 V=30.0 PL=1
MOVL C00936 V=30.0 PL=1
MOVL C00937 V=30.0 PL=1
MOVL C00938 V=30.0 PL=1
MOVL C00939 V=30.0 PL=1
MOVL C00940 V=30.0 PL=1
MOVL C00941 V=30.0 PL=1
MOVL C00942 V=30.0 PL=1
MOVL C00943 V=30.0 PL=1
MOVL C00944 V=30.0 PL=1
MOVL C00945 V=30.0 PL=1
MOVL C00946 V=30.0 PL=1
MOVL C00947 V=30.0 PL=1
MOVL C00948 V=30.0 PL=1
MOVL C00949 V=30.0 PL=1
MOVL C00950 V=30.0 PL=1
MOVL C00951 V=30.0 PL=1
MOVL C00952 V=30.0 PL=1
MOVL C00953 V=30.0 PL=1
MOVL C00954 V=30.0 PL=1
MOVL C00955 V=30.0 PL=1
MOVL C00956 V=30.0 PL=1
MOVL C00957 V=30.0 PL=1
MOVL C00958 V=30.0 PL=1
MOVL C00959 V=30.0 PL=1
MOVL C00960 V=30.0 PL=1
MOVL C00961 V=30.0 PL=1
MOVL C00962 V=30.0 PL=1
MOVL C00963 V=30.0 PL=1
MOVL C00964 V=30.0 PL=1
MOVL C00965 V=30.0 PL=1
MOVL C00966 V=30.0 PL=1
MOVL C00967 V=30.0 PL=1
MOVL C00968 V=30.0 PL=1
MOVL C00969 V=30.0 PL=1
MOVL C00970 V=30.0 PL=1
MOVL C00971 V=30.0 PL=1
MOVL C00972 V=30.0 PL=1
MOVL C00973 V=30.0 PL=1
MOVL C00974 V=30.0 PL=1
MOVL C00975 V=30.0 PL=1
MOVL C00976 V=30.0 PL=1
MOVL C00977 V=30.0 PL=1
MOVL C00978 V=30.0 PL=1
MOVL C00979 V=30.0 PL=1
MOVL C00980 V=130.0 PL=1
MOVL C00981 V=130.0 PL=1
MOVL C00982 V=30.0 PL=1
MOVL C00983 V=30.0 PL=1
MOVL C00984 V=30.0 PL=1
END
